LIN {X 0,Y 153.008,Z 595.327,A -85,B 0,C 180,E1 -24135.997,E2 -24135.997} C_VEL
LIN {X 0,Y 157.01,Z 598.55,A -85,B 0,C 180,E1 -24140.983,E2 -24140.983} C_VEL
LIN {X 0,Y 162.458,Z 600.625,A -85,B 0,C 180,E1 -24145.633,E2 -24145.633} C_VEL
LIN {X 0,Y 169.132,Z 601.557,A -85,B 0,C 180,E1 -24149.91,E2 -24149.91} C_VEL
LIN {X 0,Y 176.931,Z 601.358,A -85,B 0,C 180,E1 -24153.787,E2 -24153.787} C_VEL
LIN {X 0,Y 185.752,Z 600.036,A -85,B 0,C 180,E1 -24157.255,E2 -24157.255} C_VEL
LIN {X 0,Y 195.529,Z 597.531,A -85,B 0,C 180,E1 -24160.314,E2 -24160.314} C_VEL
LIN {X 0,Y 197.725,Z 596.972,A -85,B 0,C 180,E1 -24161.717,E2 -24161.717} C_VEL
LIN {X 0,Y 197.721,Z 597.127,A -85,B 0,C 180,E1 -24162.481,E2 -24162.481} C_VEL
LIN {X 0,Y 196.64,Z 597.978,A -85,B 0,C 180,E1 -24164.372,E2 -24164.372} C_VEL
LIN {X 0,Y 193.625,Z 599.675,A -85,B 0,C 180,E1 -24166.398,E2 -24166.398} C_VEL
LIN {X 0,Y 192.66,Z 600.123,A -85,B 0,C 180,E1 -24166.851,E2 -24166.851} C_VEL
LIN {X 0,Y 184.258,Z 603.417,A -85,B 0,C 180,E1 -24169.577,E2 -24169.577} C_VEL
LIN {X 0,Y 175.235,Z 606.225,A -85,B 0,C 180,E1 -24173.015,E2 -24173.015} C_VEL
LIN {X 0,Y 167.435,Z 608.021,A -85,B 0,C 180,E1 -24176.929,E2 -24176.929} C_VEL
LIN {X 0,Y 160.889,Z 608.807,A -85,B 0,C 180,E1 -24181.281,E2 -24181.281} C_VEL
LIN {X 0,Y 155.776,Z 608.587,A -85,B 0,C 180,E1 -24186.043,E2 -24186.043} C_VEL
LIN {X 0,Y 151.98,Z 607.326,A -85,B 0,C 180,E1 -24191.113,E2 -24191.113} C_VEL
LIN {X 0,Y 149.998,Z 605.016,A -85,B 0,C 180,E1 -24196.451,E2 -24196.451} C_VEL
LIN {X 0,Y 149.476,Z 601.54,A -85,B 0,C 180,E1 -24201.891,E2 -24201.891} C_VEL
LIN {X 0,Y 150.246,Z 596.672,A -85,B 0,C 180,E1 -24207.319,E2 -24207.319} C_VEL
LIN {X 0,Y 150.489,Z 593.443,A -85,B 0,C 180,E1 -24210,E2 -24210} C_VEL
LIN {X 0,Y 150.474,Z 587.289,A -85,B 0,C 180,E1 -24214.017,E2 -24214.017} C_VEL
LIN {X 0,Y 150.541,Z 579.575,A -85,B 0,C 180,E1 -24218.051,E2 -24218.051} C_VEL
LIN {X 0,Y 151.009,Z 570.809,A -85,B 0,C 180,E1 -24221.807,E2 -24221.807} C_VEL
LIN {X 0,Y 151.993,Z 560.329,A -85,B 0,C 180,E1 -24225.419,E2 -24225.419} C_VEL
LIN {X 0,Y 152.344,Z 554.548,A -85,B 0,C 180,E1 -24227.103,E2 -24227.103} C_VEL
LIN {X 0,Y 150.807,Z 542.716,A -85,B 0,C 180,E1 -24229.913,E2 -24229.913} C_VEL
LIN {X 0,Y 149.592,Z 528.841,A -85,B 0,C 180,E1 -24232.622,E2 -24232.622} C_VEL
LIN {X 0,Y 149.049,Z 513.657,A -85,B 0,C 180,E1 -24234.924,E2 -24234.924} C_VEL
LIN {X 0,Y 149.125,Z 509.454,A -85,B 0,C 180,E1 -24235.449,E2 -24235.449} C_VEL
LIN {X 0,Y 150.143,Z 505.621,A -85,B 0,C 180,E1 -24240.99,E2 -24240.99} C_VEL
LIN {X 0,Y 151.273,Z 502.439,A -85,B 0,C 180,E1 -24245.531,E2 -24245.531} C_VEL
LIN {X 0,Y 151.527,Z 500.732,A -85,B 0,C 180,E1 -24247.957,E2 -24247.957} C_VEL
LIN {X 0,Y 150.881,Z 497.692,A -85,B 0,C 180,E1 -24252.599,E2 -24252.599} C_VEL
LIN {X 0,Y 150.453,Z 497.743,A -85,B 0,C 180,E1 -24254.085,E2 -24254.085} C_VEL
LIN {X 0,Y 148.952,Z 497.931,A -85,B 0,C 180,E1 -24256.277,E2 -24256.277} C_VEL
LIN {X 0,Y 143.472,Z 498.608,A -85,B 0,C 180,E1 -24263.01,E2 -24263.01} C_VEL
LIN {X 0,Y 143.122,Z 498.65,A -85,B 0,C 180,E1 -24264.606,E2 -24264.606} C_VEL
LIN {X 0,Y 143.186,Z 498.648,A -85,B 0,C 180,E1 -24267.323,E2 -24267.323} C_VEL
LIN {X 0,Y 143.19,Z 498.642,A -85,B 0,C 180,E1 -24272.063,E2 -24272.063} C_VEL
LIN {X 0,Y 143.278,Z 498.634,A -85,B 0,C 180,E1 -24278.745,E2 -24278.745} C_VEL
LIN {X 0,Y 143.324,Z 498.632,A -85,B 0,C 180,E1 -24282.89,E2 -24282.89} C_VEL
LIN {X 0,Y 143.603,Z 498.591,A -85,B 0,C 180,E1 -24288.711,E2 -24288.711} C_VEL
LIN {X 0,Y 143.686,Z 498.585,A -85,B 0,C 180,E1 -24291.563,E2 -24291.563} C_VEL
LIN {X 0,Y 144.179,Z 498.523,A -85,B 0,C 180,E1 -24300,E2 -24300} C_VEL
LIN {X 0,Y 143.686,Z 498.584,A -85,B 0,C 180,E1 -24308.438,E2 -24308.438} C_VEL
LIN {X 0,Y 143.572,Z 498.6,A -85,B 0,C 180,E1 -24311.758,E2 -24311.758} C_VEL
LIN {X 0,Y 143.307,Z 498.631,A -85,B 0,C 180,E1 -24317.113,E2 -24317.113} C_VEL
LIN {X 0,Y 143.278,Z 498.636,A -85,B 0,C 180,E1 -24321.255,E2 -24321.255} C_VEL
LIN {X 0,Y 143.192,Z 498.648,A -85,B 0,C 180,E1 -24327.938,E2 -24327.938} C_VEL
LIN {X 0,Y 143.145,Z 498.647,A -85,B 0,C 180,E1 -24333.421,E2 -24333.421} C_VEL
LIN {X 0,Y 143.062,Z 498.663,A -85,B 0,C 180,E1 -24339.691,E2 -24339.691} C_VEL
LIN {X 0,Y 143.057,Z 498.661,A -85,B 0,C 180,E1 -24343.456,E2 -24343.456} C_VEL
LIN {X 0,Y 143.069,Z 498.662,A -85,B 0,C 180,E1 -24347.465,E2 -24347.465} C_VEL
LIN {X 0,Y 143.108,Z 498.654,A -85,B 0,C 180,E1 -24351.792,E2 -24351.792} C_VEL
LIN {X 0,Y 143.188,Z 498.646,A -85,B 0,C 180,E1 -24357.323,E2 -24357.323} C_VEL
LIN {X 0,Y 143.193,Z 498.647,A -85,B 0,C 180,E1 -24362.063,E2 -24362.063} C_VEL
LIN {X 0,Y 143.28,Z 498.633,A -85,B 0,C 180,E1 -24368.746,E2 -24368.746} C_VEL
LIN {X 0,Y 143.305,Z 498.633,A -85,B 0,C 180,E1 -24372.887,E2 -24372.887} C_VEL
LIN {X 0,Y 143.54,Z 498.603,A -85,B 0,C 180,E1 -24378.706,E2 -24378.706} C_VEL
LIN {X 0,Y 143.627,Z 498.594,A -85,B 0,C 180,E1 -24381.559,E2 -24381.559} C_VEL
LIN {X 0,Y 144.179,Z 498.527,A -85,B 0,C 180,E1 -24390,E2 -24390} C_VEL
LIN {X 0,Y 143.63,Z 498.594,A -85,B 0,C 180,E1 -24398.442,E2 -24398.442} C_VEL
LIN {X 0,Y 143.509,Z 498.606,A -85,B 0,C 180,E1 -24401.631,E2 -24401.631} C_VEL
LIN {X 0,Y 143.305,Z 498.633,A -85,B 0,C 180,E1 -24407.113,E2 -24407.113} C_VEL
LIN {X 0,Y 143.28,Z 498.633,A -85,B 0,C 180,E1 -24411.255,E2 -24411.255} C_VEL
LIN {X 0,Y 143.194,Z 498.647,A -85,B 0,C 180,E1 -24417.938,E2 -24417.938} C_VEL
LIN {X 0,Y 143.172,Z 498.649,A -85,B 0,C 180,E1 -24423.436,E2 -24423.436} C_VEL
LIN {X 0,Y 143.078,Z 498.657,A -85,B 0,C 180,E1 -24429.685,E2 -24429.685} C_VEL
LIN {X 0,Y 143.059,Z 498.665,A -85,B 0,C 180,E1 -24433.454,E2 -24433.454} C_VEL
LIN {X 0,Y 143.019,Z 498.665,A -85,B 0,C 180,E1 -24437.486,E2 -24437.486} C_VEL
LIN {X 0,Y 142.933,Z 498.682,A -85,B 0,C 180,E1 -24441.881,E2 -24441.881} C_VEL
LIN {X 0,Y 142.658,Z 498.708,A -85,B 0,C 180,E1 -24447.185,E2 -24447.185} C_VEL
LIN {X 0,Y 142.204,Z 498.771,A -85,B 0,C 180,E1 -24453.589,E2 -24453.589} C_VEL
LIN {X 0,Y 142.169,Z 498.848,A -85,B 0,C 180,E1 -24455.785,E2 -24455.785} C_VEL
LIN {X 0,Y 144.366,Z 512.297,A -85,B 0,C 180,E1 -24457.963,E2 -24457.963} C_VEL
LIN {X 0,Y 146.228,Z 522.624,A -85,B 0,C 180,E1 -24459.99,E2 -24459.99} C_VEL
LIN {X 0,Y 146.161,Z 525.789,A -85,B 0,C 180,E1 -24460.696,E2 -24460.696} C_VEL
LIN {X 0,Y 144.531,Z 538.8,A -85,B 0,C 180,E1 -24464.125,E2 -24464.125} C_VEL
LIN {X 0,Y 143.248,Z 550.554,A -85,B 0,C 180,E1 -24467.964,E2 -24467.964} C_VEL
LIN {X 0,Y 142.27,Z 561.149,A -85,B 0,C 180,E1 -24472.268,E2 -24472.268} C_VEL
LIN {X 0,Y 141.759,Z 570.856,A -85,B 0,C 180,E1 -24477.158,E2 -24477.158} C_VEL
LIN {X 0,Y 141.689,Z 577.811,A -85,B 0,C 180,E1 -24481.421,E2 -24481.421} C_VEL
LIN {X 0,Y 142.098,Z 583.58,A -85,B 0,C 180,E1 -24485.676,E2 -24485.676} C_VEL
LIN {X 0,Y 143.502,Z 590.092,A -85,B 0,C 180,E1 -24491.619,E2 -24491.619} C_VEL
LIN {X 0,Y 146.244,Z 594.625,A -85,B 0,C 180,E1 -24496.758,E2 -24496.758} C_VEL
LIN {X 0,Y 150.409,Z 598.253,A -85,B 0,C 180,E1 -24501.95,E2 -24501.95} C_VEL
LIN {X 0,Y 156.095,Z 600.718,A -85,B 0,C 180,E1 -24506.759,E2 -24506.759} C_VEL
LIN {X 0,Y 163.032,Z 602.071,A -85,B 0,C 180,E1 -24511.151,E2 -24511.151} C_VEL
LIN {X 0,Y 171.146,Z 602.303,A -85,B 0,C 180,E1 -24515.093,E2 -24515.093} C_VEL
LIN {X 0,Y 180.244,Z 601.445,A -85,B 0,C 180,E1 -24518.599,E2 -24518.599} C_VEL
LIN {X 0,Y 190.21,Z 599.482,A -85,B 0,C 180,E1 -24521.688,E2 -24521.688} C_VEL
LIN {X 0,Y 190.811,Z 599.467,A -85,B 0,C 180,E1 -24522.553,E2 -24522.553} C_VEL
LIN {X 0,Y 188.352,Z 600.781,A -85,B 0,C 180,E1 -24524.85,E2 -24524.85} C_VEL
LIN {X 0,Y 183.913,Z 602.443,A -85,B 0,C 180,E1 -24526.54,E2 -24526.54} C_VEL
LIN {X 0,Y 174.157,Z 605.288,A -85,B 0,C 180,E1 -24529.784,E2 -24529.784} C_VEL
LIN {X 0,Y 165.429,Z 607.134,A -85,B 0,C 180,E1 -24533.503,E2 -24533.503} C_VEL
LIN {X 0,Y 157.935,Z 608.004,A -85,B 0,C 180,E1 -24537.724,E2 -24537.724} C_VEL
LIN {X 0,Y 151.845,Z 607.905,A -85,B 0,C 180,E1 -24542.429,E2 -24542.429} C_VEL
LIN {X 0,Y 147.187,Z 606.83,A -85,B 0,C 180,E1 -24547.543,E2 -24547.543} C_VEL
LIN {X 0,Y 144.13,Z 604.743,A -85,B 0,C 180,E1 -24552.988,E2 -24552.988} C_VEL
LIN {X 0,Y 142.804,Z 601.556,A -85,B 0,C 180,E1 -24558.646,E2 -24558.646} C_VEL
LIN {X 0,Y 142.978,Z 597.154,A -85,B 0,C 180,E1 -24564.358,E2 -24564.358} C_VEL
LIN {X 0,Y 143.527,Z 594.379,A -85,B 0,C 180,E1 -24567.193,E2 -24567.193} C_VEL
LIN {X 0,Y 143.742,Z 590.953,A -85,B 0,C 180,E1 -24570,E2 -24570} C_VEL
LIN {X 0,Y 143.679,Z 585.695,A -85,B 0,C 180,E1 -24573.505,E2 -24573.505} C_VEL
LIN {X 0,Y 143.696,Z 579.205,A -85,B 0,C 180,E1 -24577.023,E2 -24577.023} C_VEL
LIN {X 0,Y 144.117,Z 569.784,A -85,B 0,C 180,E1 -24581.248,E2 -24581.248} C_VEL
LIN {X 0,Y 145.163,Z 558.179,A -85,B 0,C 180,E1 -24585.443,E2 -24585.443} C_VEL
LIN {X 0,Y 145.4,Z 554.724,A -85,B 0,C 180,E1 -24586.497,E2 -24586.497} C_VEL
LIN {X 0,Y 143.724,Z 542.198,A -85,B 0,C 180,E1 -24589.644,E2 -24589.644} C_VEL
LIN {X 0,Y 142.532,Z 529.062,A -85,B 0,C 180,E1 -24592.361,E2 -24592.361} C_VEL
LIN {X 0,Y 141.964,Z 514.809,A -85,B 0,C 180,E1 -24594.689,E2 -24594.689} C_VEL
LIN {X 0,Y 142.057,Z 508.996,A -85,B 0,C 180,E1 -24595.553,E2 -24595.553} C_VEL
LIN {X 0,Y 143.396,Z 504.379,A -85,B 0,C 180,E1 -24602.624,E2 -24602.624} C_VEL
LIN {X 0,Y 144.212,Z 502.265,A -85,B 0,C 180,E1 -24605.789,E2 -24605.789} C_VEL
LIN {X 0,Y 144.426,Z 501.307,A -85,B 0,C 180,E1 -24607.224,E2 -24607.224} C_VEL
LIN {X 0,Y 143.911,Z 498.562,A -85,B 0,C 180,E1 -24611.532,E2 -24611.532} C_VEL
LIN {X 0,Y 143.428,Z 498.618,A -85,B 0,C 180,E1 -24617.307,E2 -24617.307} C_VEL
LIN {X 0,Y 143.146,Z 498.649,A -85,B 0,C 180,E1 -24623.903,E2 -24623.903} C_VEL
LIN {X 0,Y 143.122,Z 498.65,A -85,B 0,C 180,E1 -24624.606,E2 -24624.606} C_VEL
LIN {X 0,Y 142.413,Z 498.746,A -85,B 0,C 180,E1 -24626.956,E2 -24626.956} C_VEL
LIN {X 0,Y 140.803,Z 498.943,A -85,B 0,C 180,E1 -24629.272,E2 -24629.272} C_VEL
LIN {X 0,Y 137.111,Z 499.403,A -85,B 0,C 180,E1 -24634.004,E2 -24634.004} C_VEL
LIN {X 0,Y 136.163,Z 499.525,A -85,B 0,C 180,E1 -24636.497,E2 -24636.497} C_VEL
LIN {X 0,Y 136.127,Z 499.523,A -85,B 0,C 180,E1 -24637.341,E2 -24637.341} C_VEL
LIN {X 0,Y 136.258,Z 499.508,A -85,B 0,C 180,E1 -24641.973,E2 -24641.973} C_VEL
LIN {X 0,Y 136.502,Z 499.477,A -85,B 0,C 180,E1 -24648.116,E2 -24648.116} C_VEL
LIN {X 0,Y 136.61,Z 499.467,A -85,B 0,C 180,E1 -24651.122,E2 -24651.122} C_VEL
LIN {X 0,Y 137.136,Z 499.4,A -85,B 0,C 180,E1 -24660.001,E2 -24660.001} C_VEL
LIN {X 0,Y 136.61,Z 499.467,A -85,B 0,C 180,E1 -24668.879,E2 -24668.879} C_VEL
LIN {X 0,Y 136.493,Z 499.483,A -85,B 0,C 180,E1 -24671.957,E2 -24671.957} C_VEL
LIN {X 0,Y 136.246,Z 499.512,A -85,B 0,C 180,E1 -24678.03,E2 -24678.03} C_VEL
LIN {X 0,Y 136.199,Z 499.518,A -85,B 0,C 180,E1 -24681.75,E2 -24681.75} C_VEL
LIN {X 0,Y 136.118,Z 499.53,A -85,B 0,C 180,E1 -24688.629,E2 -24688.629} C_VEL
LIN {X 0,Y 136.044,Z 499.536,A -85,B 0,C 180,E1 -24694.63,E2 -24694.63} C_VEL
LIN {X 0,Y 136.033,Z 499.538,A -85,B 0,C 180,E1 -24699.199,E2 -24699.199} C_VEL
LIN {X 0,Y 135.999,Z 499.541,A -85,B 0,C 180,E1 -24703.658,E2 -24703.658} C_VEL
LIN {X 0,Y 136.033,Z 499.54,A -85,B 0,C 180,E1 -24707.807,E2 -24707.807} C_VEL
LIN {X 0,Y 136.057,Z 499.532,A -85,B 0,C 180,E1 -24711.695,E2 -24711.695} C_VEL
LIN {X 0,Y 136.092,Z 499.533,A -85,B 0,C 180,E1 -24715.718,E2 -24715.718} C_VEL
LIN {X 0,Y 136.149,Z 499.526,A -85,B 0,C 180,E1 -24722.317,E2 -24722.317} C_VEL
LIN {X 0,Y 136.247,Z 499.509,A -85,B 0,C 180,E1 -24728.834,E2 -24728.834} C_VEL
LIN {X 0,Y 136.272,Z 499.507,A -85,B 0,C 180,E1 -24735.057,E2 -24735.057} C_VEL
LIN {X 0,Y 136.447,Z 499.484,A -85,B 0,C 180,E1 -24738.138,E2 -24738.138} C_VEL
LIN {X 0,Y 136.553,Z 499.475,A -85,B 0,C 180,E1 -24741.118,E2 -24741.118} C_VEL
LIN {X 0,Y 137.136,Z 499.404,A -85,B 0,C 180,E1 -24750,E2 -24750} C_VEL
LIN {X 0,Y 136.555,Z 499.474,A -85,B 0,C 180,E1 -24758.882,E2 -24758.882} C_VEL
LIN {X 0,Y 136.444,Z 499.484,A -85,B 0,C 180,E1 -24761.89,E2 -24761.89} C_VEL
LIN {X 0,Y 136.246,Z 499.514,A -85,B 0,C 180,E1 -24768.03,E2 -24768.03} C_VEL
LIN {X 0,Y 136.201,Z 499.513,A -85,B 0,C 180,E1 -24771.749,E2 -24771.749} C_VEL
LIN {X 0,Y 136.104,Z 499.528,A -85,B 0,C 180,E1 -24778.617,E2 -24778.617} C_VEL
LIN {X 0,Y 136.082,Z 499.533,A -85,B 0,C 180,E1 -24784.618,E2 -24784.618} C_VEL
LIN {X 0,Y 136.053,Z 499.532,A -85,B 0,C 180,E1 -24789.208,E2 -24789.208} C_VEL
LIN {X 0,Y 135.999,Z 499.545,A -85,B 0,C 180,E1 -24793.657,E2 -24793.657} C_VEL
LIN {X 0,Y 135.961,Z 499.543,A -85,B 0,C 180,E1 -24797.779,E2 -24797.779} C_VEL
LIN {X 0,Y 135.888,Z 499.558,A -85,B 0,C 180,E1 -24801.637,E2 -24801.637} C_VEL
LIN {X 0,Y 135.657,Z 499.581,A -85,B 0,C 180,E1 -24805.988,E2 -24805.988} C_VEL
LIN {X 0,Y 135.188,Z 499.647,A -85,B 0,C 180,E1 -24812.102,E2 -24812.102} C_VEL
LIN {X 0,Y 135.129,Z 499.65,A -85,B 0,C 180,E1 -24815.897,E2 -24815.897} C_VEL
LIN {X 0,Y 137.922,Z 516.294,A -85,B 0,C 180,E1 -24818.882,E2 -24818.882} C_VEL
LIN {X 0,Y 139.254,Z 523.712,A -85,B 0,C 180,E1 -24820.466,E2 -24820.466} C_VEL
LIN {X 0,Y 137.75,Z 536.019,A -85,B 0,C 180,E1 -24823.703,E2 -24823.703} C_VEL
LIN {X 0,Y 136.451,Z 547.152,A -85,B 0,C 180,E1 -24827.355,E2 -24827.355} C_VEL
LIN {X 0,Y 135.402,Z 558.315,A -85,B 0,C 180,E1 -24831.873,E2 -24831.873} C_VEL
LIN {X 0,Y 134.91,Z 567.261,A -85,B 0,C 180,E1 -24836.266,E2 -24836.266} C_VEL
LIN {X 0,Y 134.818,Z 573.635,A -85,B 0,C 180,E1 -24839.999,E2 -24839.999} C_VEL
LIN {X 0,Y 135.041,Z 580.054,A -85,B 0,C 180,E1 -24844.477,E2 -24844.477} C_VEL
LIN {X 0,Y 135.991,Z 586.675,A -85,B 0,C 180,E1 -24850.019,E2 -24850.019} C_VEL
LIN {X 0,Y 138.585,Z 592.587,A -85,B 0,C 180,E1 -24856.195,E2 -24856.195} C_VEL
LIN {X 0,Y 141.542,Z 595.948,A -85,B 0,C 180,E1 -24860.339,E2 -24860.339} C_VEL
LIN {X 0,Y 146.668,Z 599.355,A -85,B 0,C 180,E1 -24865.547,E2 -24865.547} C_VEL
LIN {X 0,Y 153.253,Z 601.654,A -85,B 0,C 180,E1 -24870.294,E2 -24870.294} C_VEL
LIN {X 0,Y 161.114,Z 602.867,A -85,B 0,C 180,E1 -24874.546,E2 -24874.546} C_VEL
LIN {X 0,Y 170.016,Z 602.999,A -85,B 0,C 180,E1 -24878.32,E2 -24878.32} C_VEL
LIN {X 0,Y 179.888,Z 602.056,A -85,B 0,C 180,E1 -24881.618,E2 -24881.618} C_VEL
LIN {X 0,Y 182.895,Z 601.722,A -85,B 0,C 180,E1 -24883.104,E2 -24883.104} C_VEL
LIN {X 0,Y 178.839,Z 603.077,A -85,B 0,C 180,E1 -24884.979,E2 -24884.979} C_VEL
LIN {X 0,Y 168.804,Z 605.434,A -85,B 0,C 180,E1 -24888.229,E2 -24888.229} C_VEL
LIN {X 0,Y 159.802,Z 606.846,A -85,B 0,C 180,E1 -24891.996,E2 -24891.996} C_VEL
LIN {X 0,Y 151.763,Z 607.311,A -85,B 0,C 180,E1 -24896.466,E2 -24896.466} C_VEL
LIN {X 0,Y 145.644,Z 606.854,A -85,B 0,C 180,E1 -24901.148,E2 -24901.148} C_VEL
LIN {X 0,Y 140.773,Z 605.448,A -85,B 0,C 180,E1 -24906.459,E2 -24906.459} C_VEL
LIN {X 0,Y 137.543,Z 603.026,A -85,B 0,C 180,E1 -24912.146,E2 -24912.146} C_VEL
LIN {X 0,Y 136.054,Z 598.966,A -85,B 0,C 180,E1 -24918.949,E2 -24918.949} C_VEL
LIN {X 0,Y 136.299,Z 594.862,A -85,B 0,C 180,E1 -24924.08,E2 -24924.08} C_VEL
LIN {X 0,Y 136.862,Z 591.94,A -85,B 0,C 180,E1 -24927.056,E2 -24927.056} C_VEL
LIN {X 0,Y 137.023,Z 588.289,A -85,B 0,C 180,E1 -24930,E2 -24930} C_VEL
LIN {X 0,Y 136.982,Z 582.68,A -85,B 0,C 180,E1 -24933.677,E2 -24933.677} C_VEL
LIN {X 0,Y 136.988,Z 574.415,A -85,B 0,C 180,E1 -24938.11,E2 -24938.11} C_VEL
LIN {X 0,Y 137.403,Z 565.912,A -85,B 0,C 180,E1 -24941.806,E2 -24941.806} C_VEL
LIN {X 0,Y 138.405,Z 554.702,A -85,B 0,C 180,E1 -24945.8,E2 -24945.8} C_VEL
LIN {X 0,Y 136.981,Z 543.992,A -85,B 0,C 180,E1 -24948.703,E2 -24948.703} C_VEL
LIN {X 0,Y 135.712,Z 531.069,A -85,B 0,C 180,E1 -24951.612,E2 -24951.612} C_VEL
LIN {X 0,Y 134.973,Z 518,A -85,B 0,C 180,E1 -24954.003,E2 -24954.003} C_VEL
LIN {X 0,Y 134.986,Z 508.64,A -85,B 0,C 180,E1 -24955.438,E2 -24955.438} C_VEL
LIN {X 0,Y 136.32,Z 504.122,A -85,B 0,C 180,E1 -24962.774,E2 -24962.774} C_VEL
LIN {X 0,Y 137.173,Z 502.018,A -85,B 0,C 180,E1 -24966.138,E2 -24966.138} C_VEL
LIN {X 0,Y 137.245,Z 500.905,A -85,B 0,C 180,E1 -24967.915,E2 -24967.915} C_VEL
LIN {X 0,Y 136.935,Z 499.431,A -85,B 0,C 180,E1 -24970.407,E2 -24970.407} C_VEL
LIN {X 0,Y 136.452,Z 499.488,A -85,B 0,C 180,E1 -24976.143,E2 -24976.143} C_VEL
LIN {X 0,Y 136.167,Z 499.518,A -85,B 0,C 180,E1 -24981.731,E2 -24981.731} C_VEL
LIN {X 0,Y 136.096,Z 499.531,A -85,B 0,C 180,E1 -24985.714,E2 -24985.714} C_VEL
LIN {X 0,Y 136.146,Z 499.52,A -85,B 0,C 180,E1 -24992.317,E2 -24992.317} C_VEL
LIN {X 0,Y 136.127,Z 499.523,A -85,B 0,C 180,E1 -24997.341,E2 -24997.341} C_VEL
LIN {X 0,Y 135.629,Z 499.591,A -85,B 0,C 180,E1 -24999.812,E2 -24999.812} C_VEL
LIN {X 0,Y 134.228,Z 499.773,A -85,B 0,C 180,E1 -25002.258,E2 -25002.258} C_VEL
LIN {X 0,Y 129.908,Z 500.307,A -85,B 0,C 180,E1 -25008.981,E2 -25008.981} C_VEL
LIN {X 0,Y 129.524,Z 500.346,A -85,B 0,C 180,E1 -25010.752,E2 -25010.752} C_VEL
LIN {X 0,Y 130.091,Z 500.277,A -85,B 0,C 180,E1 -25020.001,E2 -25020.001} C_VEL
LIN {X 0,Y 129.532,Z 500.348,A -85,B 0,C 180,E1 -25029.368,E2 -25029.368} C_VEL
LIN {X 0,Y 129.394,Z 500.366,A -85,B 0,C 180,E1 -25032.549,E2 -25032.549} C_VEL
LIN {X 0,Y 129.157,Z 500.396,A -85,B 0,C 180,E1 -25039.056,E2 -25039.056} C_VEL
LIN {X 0,Y 129.109,Z 500.399,A -85,B 0,C 180,E1 -25042.399,E2 -25042.399} C_VEL
LIN {X 0,Y 129.037,Z 500.411,A -85,B 0,C 180,E1 -25049.374,E2 -25049.374} C_VEL
LIN {X 0,Y 128.96,Z 500.419,A -85,B 0,C 180,E1 -25055.169,E2 -25055.169} C_VEL
LIN {X 0,Y 128.935,Z 500.418,A -85,B 0,C 180,E1 -25060.852,E2 -25060.852} C_VEL
LIN {X 0,Y 128.923,Z 500.425,A -85,B 0,C 180,E1 -25065.128,E2 -25065.128} C_VEL
LIN {X 0,Y 128.959,Z 500.416,A -85,B 0,C 180,E1 -25069.728,E2 -25069.728} C_VEL
LIN {X 0,Y 128.994,Z 500.416,A -85,B 0,C 180,E1 -25074.811,E2 -25074.811} C_VEL
LIN {X 0,Y 129.036,Z 500.408,A -85,B 0,C 180,E1 -25080.647,E2 -25080.647} C_VEL
LIN {X 0,Y 129.111,Z 500.396,A -85,B 0,C 180,E1 -25087.602,E2 -25087.602} C_VEL
LIN {X 0,Y 129.156,Z 500.395,A -85,B 0,C 180,E1 -25090.945,E2 -25090.945} C_VEL
LIN {X 0,Y 129.369,Z 500.364,A -85,B 0,C 180,E1 -25097.923,E2 -25097.923} C_VEL
LIN {X 0,Y 129.479,Z 500.356,A -85,B 0,C 180,E1 -25100.629,E2 -25100.629} C_VEL
LIN {X 0,Y 130.091,Z 500.281,A -85,B 0,C 180,E1 -25110,E2 -25110} C_VEL
LIN {X 0,Y 129.481,Z 500.356,A -85,B 0,C 180,E1 -25119.372,E2 -25119.372} C_VEL
LIN {X 0,Y 129.347,Z 500.366,A -85,B 0,C 180,E1 -25122.553,E2 -25122.553} C_VEL
LIN {X 0,Y 129.157,Z 500.395,A -85,B 0,C 180,E1 -25129.056,E2 -25129.056} C_VEL
LIN {X 0,Y 129.111,Z 500.396,A -85,B 0,C 180,E1 -25132.398,E2 -25132.398} C_VEL
LIN {X 0,Y 129.039,Z 500.408,A -85,B 0,C 180,E1 -25139.373,E2 -25139.373} C_VEL
LIN {X 0,Y 128.995,Z 500.416,A -85,B 0,C 180,E1 -25145.189,E2 -25145.189} C_VEL
LIN {X 0,Y 128.953,Z 500.417,A -85,B 0,C 180,E1 -25150.845,E2 -25150.845} C_VEL
LIN {X 0,Y 128.915,Z 500.426,A -85,B 0,C 180,E1 -25155.131,E2 -25155.131} C_VEL
LIN {X 0,Y 128.851,Z 500.43,A -85,B 0,C 180,E1 -25159.784,E2 -25159.784} C_VEL
LIN {X 0,Y 128.641,Z 500.459,A -85,B 0,C 180,E1 -25165.035,E2 -25165.035} C_VEL
LIN {X 0,Y 128.18,Z 500.518,A -85,B 0,C 180,E1 -25171.315,E2 -25171.315} C_VEL
LIN {X 0,Y 128.1,Z 500.545,A -85,B 0,C 180,E1 -25176.176,E2 -25176.176} C_VEL
LIN {X 0,Y 130.435,Z 514.22,A -85,B 0,C 180,E1 -25178.672,E2 -25178.672} C_VEL
LIN {X 0,Y 132.042,Z 522.98,A -85,B 0,C 180,E1 -25180.569,E2 -25180.569} C_VEL
LIN {X 0,Y 130.886,Z 534.1,A -85,B 0,C 180,E1 -25183.626,E2 -25183.626} C_VEL
LIN {X 0,Y 129.473,Z 546.18,A -85,B 0,C 180,E1 -25187.709,E2 -25187.709} C_VEL
LIN {X 0,Y 128.466,Z 557.428,A -85,B 0,C 180,E1 -25192.418,E2 -25192.418} C_VEL
LIN {X 0,Y 128.043,Z 566.099,A -85,B 0,C 180,E1 -25196.853,E2 -25196.853} C_VEL
LIN {X 0,Y 127.958,Z 572.573,A -85,B 0,C 180,E1 -25200.786,E2 -25200.786} C_VEL
LIN {X 0,Y 128.341,Z 580.211,A -85,B 0,C 180,E1 -25206.287,E2 -25206.287} C_VEL
LIN {X 0,Y 129.764,Z 587.161,A -85,B 0,C 180,E1 -25212.511,E2 -25212.511} C_VEL
LIN {X 0,Y 132.846,Z 592.772,A -85,B 0,C 180,E1 -25218.507,E2 -25218.507} C_VEL
LIN {X 0,Y 137.388,Z 597.118,A -85,B 0,C 180,E1 -25224.156,E2 -25224.156} C_VEL
LIN {X 0,Y 143.57,Z 600.352,A -85,B 0,C 180,E1 -25229.309,E2 -25229.309} C_VEL
LIN {X 0,Y 151.093,Z 602.529,A -85,B 0,C 180,E1 -25233.929,E2 -25233.929} C_VEL
LIN {X 0,Y 159.801,Z 603.643,A -85,B 0,C 180,E1 -25238.004,E2 -25238.004} C_VEL
LIN {X 0,Y 169.49,Z 603.71,A -85,B 0,C 180,E1 -25241.563,E2 -25241.563} C_VEL
LIN {X 0,Y 173.82,Z 603.52,A -85,B 0,C 180,E1 -25243.298,E2 -25243.298} C_VEL
LIN {X 0,Y 163.577,Z 605.412,A -85,B 0,C 180,E1 -25246.572,E2 -25246.572} C_VEL
LIN {X 0,Y 154.285,Z 606.384,A -85,B 0,C 180,E1 -25250.377,E2 -25250.377} C_VEL
LIN {X 0,Y 145.75,Z 606.434,A -85,B 0,C 180,E1 -25255.058,E2 -25255.058} C_VEL
LIN {X 0,Y 139.555,Z 605.644,A -85,B 0,C 180,E1 -25259.761,E2 -25259.761} C_VEL
LIN {X 0,Y 134.444,Z 603.904,A -85,B 0,C 180,E1 -25265.279,E2 -25265.279} C_VEL
LIN {X 0,Y 131.029,Z 601.2,A -85,B 0,C 180,E1 -25271.226,E2 -25271.226} C_VEL
LIN {X 0,Y 129.473,Z 597.264,A -85,B 0,C 180,E1 -25277.705,E2 -25277.705} C_VEL
LIN {X 0,Y 129.699,Z 592.413,A -85,B 0,C 180,E1 -25283.778,E2 -25283.778} C_VEL
LIN {X 0,Y 130.238,Z 589.325,A -85,B 0,C 180,E1 -25286.906,E2 -25286.906} C_VEL
LIN {X 0,Y 130.367,Z 585.481,A -85,B 0,C 180,E1 -25290,E2 -25290} C_VEL
LIN {X 0,Y 130.252,Z 579.485,A -85,B 0,C 180,E1 -25293.867,E2 -25293.867} C_VEL
LIN {X 0,Y 130.299,Z 570.655,A -85,B 0,C 180,E1 -25298.53,E2 -25298.53} C_VEL
LIN {X 0,Y 130.905,Z 559.932,A -85,B 0,C 180,E1 -25303.114,E2 -25303.114} C_VEL
LIN {X 0,Y 131.416,Z 553.21,A -85,B 0,C 180,E1 -25305.509,E2 -25305.509} C_VEL
LIN {X 0,Y 129.566,Z 540.521,A -85,B 0,C 180,E1 -25308.993,E2 -25308.993} C_VEL
LIN {X 0,Y 128.327,Z 527.464,A -85,B 0,C 180,E1 -25311.962,E2 -25311.962} C_VEL
LIN {X 0,Y 127.801,Z 513.007,A -85,B 0,C 180,E1 -25314.574,E2 -25314.574} C_VEL
LIN {X 0,Y 127.917,Z 508.243,A -85,B 0,C 180,E1 -25315.31,E2 -25315.31} C_VEL
LIN {X 0,Y 129.23,Z 503.862,A -85,B 0,C 180,E1 -25322.945,E2 -25322.945} C_VEL
LIN {X 0,Y 130.093,Z 501.79,A -85,B 0,C 180,E1 -25326.459,E2 -25326.459} C_VEL
LIN {X 0,Y 129.978,Z 500.297,A -85,B 0,C 180,E1 -25329.194,E2 -25329.194} C_VEL
LIN {X 0,Y 129.486,Z 500.354,A -85,B 0,C 180,E1 -25335.123,E2 -25335.123} C_VEL
LIN {X 0,Y 129.164,Z 500.394,A -85,B 0,C 180,E1 -25339.619,E2 -25339.619} C_VEL
LIN {X 0,Y 129.037,Z 500.409,A -85,B 0,C 180,E1 -25344.783,E2 -25344.783} C_VEL
LIN {X 0,Y 129.033,Z 500.406,A -85,B 0,C 180,E1 -25350.647,E2 -25350.647} C_VEL
LIN {X 0,Y 129.109,Z 500.401,A -85,B 0,C 180,E1 -25357.602,E2 -25357.602} C_VEL
LIN {X 0,Y 129.164,Z 500.39,A -85,B 0,C 180,E1 -25360.946,E2 -25360.946} C_VEL
LIN {X 0,Y 129.419,Z 500.36,A -85,B 0,C 180,E1 -25367.815,E2 -25367.815} C_VEL
LIN {X 0,Y 129.524,Z 500.346,A -85,B 0,C 180,E1 -25370.752,E2 -25370.752} C_VEL
LIN {X 0,Y 128.778,Z 500.445,A -85,B 0,C 180,E1 -25373.359,E2 -25373.359} C_VEL
LIN {X 0,Y 127.232,Z 500.634,A -85,B 0,C 180,E1 -25375.937,E2 -25375.937} C_VEL
LIN {X 0,Y 122.848,Z 501.182,A -85,B 0,C 180,E1 -25383.05,E2 -25383.05} C_VEL
LIN {X 0,Y 122.484,Z 501.217,A -85,B 0,C 180,E1 -25384.927,E2 -25384.927} C_VEL
LIN {X 0,Y 122.458,Z 501.23,A -85,B 0,C 180,E1 -25389.915,E2 -25389.915} C_VEL
LIN {X 0,Y 122.264,Z 501.252,A -85,B 0,C 180,E1 -25393.294,E2 -25393.294} C_VEL
LIN {X 0,Y 122.048,Z 501.283,A -85,B 0,C 180,E1 -25400.213,E2 -25400.213} C_VEL
LIN {X 0,Y 121.985,Z 501.284,A -85,B 0,C 180,E1 -25403.785,E2 -25403.785} C_VEL
LIN {X 0,Y 121.94,Z 501.295,A -85,B 0,C 180,E1 -25410.172,E2 -25410.172} C_VEL
LIN {X 0,Y 121.885,Z 501.302,A -85,B 0,C 180,E1 -25416.172,E2 -25416.172} C_VEL
LIN {X 0,Y 121.873,Z 501.297,A -85,B 0,C 180,E1 -25421.439,E2 -25421.439} C_VEL
LIN {X 0,Y 121.886,Z 501.299,A -85,B 0,C 180,E1 -25428.556,E2 -25428.556} C_VEL
LIN {X 0,Y 121.947,Z 501.294,A -85,B 0,C 180,E1 -25434.809,E2 -25434.809} C_VEL
LIN {X 0,Y 121.944,Z 501.288,A -85,B 0,C 180,E1 -25439.827,E2 -25439.827} C_VEL
LIN {X 0,Y 121.986,Z 501.286,A -85,B 0,C 180,E1 -25446.216,E2 -25446.216} C_VEL
LIN {X 0,Y 122.048,Z 501.278,A -85,B 0,C 180,E1 -25449.788,E2 -25449.788} C_VEL
LIN {X 0,Y 122.242,Z 501.25,A -85,B 0,C 180,E1 -25456.705,E2 -25456.705} C_VEL
LIN {X 0,Y 122.408,Z 501.237,A -85,B 0,C 180,E1 -25460.082,E2 -25460.082} C_VEL
LIN {X 0,Y 122.598,Z 501.209,A -85,B 0,C 180,E1 -25466.714,E2 -25466.714} C_VEL
LIN {X 0,Y 123.044,Z 501.159,A -85,B 0,C 180,E1 -25470,E2 -25470} C_VEL
LIN {X 0,Y 122.429,Z 501.233,A -85,B 0,C 180,E1 -25476.593,E2 -25476.593} C_VEL
LIN {X 0,Y 122.321,Z 501.241,A -85,B 0,C 180,E1 -25482.377,E2 -25482.377} C_VEL
LIN {X 0,Y 122.112,Z 501.273,A -85,B 0,C 180,E1 -25486.725,E2 -25486.725} C_VEL
LIN {X 0,Y 122.027,Z 501.279,A -85,B 0,C 180,E1 -25492.851,E2 -25492.851} C_VEL
LIN {X 0,Y 121.953,Z 501.294,A -85,B 0,C 180,E1 -25497.454,E2 -25497.454} C_VEL
LIN {X 0,Y 121.914,Z 501.291,A -85,B 0,C 180,E1 -25501.254,E2 -25501.254} C_VEL
LIN {X 0,Y 121.915,Z 501.298,A -85,B 0,C 180,E1 -25506.189,E2 -25506.189} C_VEL
LIN {X 0,Y 121.886,Z 501.299,A -85,B 0,C 180,E1 -25511.444,E2 -25511.444} C_VEL
LIN {X 0,Y 121.806,Z 501.309,A -85,B 0,C 180,E1 -25516.18,E2 -25516.18} C_VEL
LIN {X 0,Y 121.752,Z 501.317,A -85,B 0,C 180,E1 -25520.582,E2 -25520.582} C_VEL
LIN {X 0,Y 121.617,Z 501.334,A -85,B 0,C 180,E1 -25524.697,E2 -25524.697} C_VEL
LIN {X 0,Y 121.172,Z 501.391,A -85,B 0,C 180,E1 -25530.46,E2 -25530.46} C_VEL
LIN {X 0,Y 121.093,Z 501.398,A -85,B 0,C 180,E1 -25536.521,E2 -25536.521} C_VEL
LIN {X 0,Y 123.514,Z 515.3,A -85,B 0,C 180,E1 -25539.228,E2 -25539.228} C_VEL
LIN {X 0,Y 124.995,Z 523.585,A -85,B 0,C 180,E1 -25541.137,E2 -25541.137} C_VEL
LIN {X 0,Y 123.515,Z 535.74,A -85,B 0,C 180,E1 -25544.743,E2 -25544.743} C_VEL
LIN {X 0,Y 122.4,Z 546.454,A -85,B 0,C 180,E1 -25548.615,E2 -25548.615} C_VEL
LIN {X 0,Y 121.526,Z 557.029,A -85,B 0,C 180,E1 -25553.358,E2 -25553.358} C_VEL
LIN {X 0,Y 121.185,Z 566.212,A -85,B 0,C 180,E1 -25558.338,E2 -25558.338} C_VEL
LIN {X 0,Y 121.206,Z 573.847,A -85,B 0,C 180,E1 -25563.324,E2 -25563.324} C_VEL
LIN {X 0,Y 121.857,Z 580.191,A -85,B 0,C 180,E1 -25568.29,E2 -25568.29} C_VEL
LIN {X 0,Y 123.891,Z 587.701,A -85,B 0,C 180,E1 -25575.34,E2 -25575.34} C_VEL
LIN {X 0,Y 128.478,Z 594.055,A -85,B 0,C 180,E1 -25582.514,E2 -25582.514} C_VEL
LIN {X 0,Y 134.066,Z 598.204,A -85,B 0,C 180,E1 -25588.151,E2 -25588.151} C_VEL
LIN {X 0,Y 141.19,Z 601.312,A -85,B 0,C 180,E1 -25593.198,E2 -25593.198} C_VEL
LIN {X 0,Y 149.649,Z 603.381,A -85,B 0,C 180,E1 -25597.627,E2 -25597.627} C_VEL
LIN {X 0,Y 161.275,Z 604.523,A -85,B 0,C 180,E1 -25602.198,E2 -25602.198} C_VEL
LIN {X 0,Y 163.716,Z 604.585,A -85,B 0,C 180,E1 -25603.132,E2 -25603.132} C_VEL
LIN {X 0,Y 153.565,Z 605.571,A -85,B 0,C 180,E1 -25606.647,E2 -25606.647} C_VEL
LIN {X 0,Y 144.589,Z 605.692,A -85,B 0,C 180,E1 -25610.81,E2 -25610.81} C_VEL
LIN {X 0,Y 136.865,Z 604.967,A -85,B 0,C 180,E1 -25615.608,E2 -25615.608} C_VEL
LIN {X 0,Y 130.675,Z 603.353,A -85,B 0,C 180,E1 -25621.05,E2 -25621.05} C_VEL
LIN {X 0,Y 126.133,Z 600.791,A -85,B 0,C 180,E1 -25627.043,E2 -25627.043} C_VEL
LIN {X 0,Y 123.541,Z 597.288,A -85,B 0,C 180,E1 -25633.474,E2 -25633.474} C_VEL
LIN {X 0,Y 122.842,Z 592.657,A -85,B 0,C 180,E1 -25640.117,E2 -25640.117} C_VEL
LIN {X 0,Y 123.394,Z 588.231,A -85,B 0,C 180,E1 -25645.099,E2 -25645.099} C_VEL
LIN {X 0,Y 123.768,Z 584.586,A -85,B 0,C 180,E1 -25648.373,E2 -25648.373} C_VEL
LIN {X 0,Y 123.641,Z 578.812,A -85,B 0,C 180,E1 -25652.443,E2 -25652.443} C_VEL
LIN {X 0,Y 123.531,Z 570.069,A -85,B 0,C 180,E1 -25657.354,E2 -25657.354} C_VEL
LIN {X 0,Y 123.886,Z 561.188,A -85,B 0,C 180,E1 -25661.452,E2 -25661.452} C_VEL
LIN {X 0,Y 124.498,Z 552.405,A -85,B 0,C 180,E1 -25664.844,E2 -25664.844} C_VEL
LIN {X 0,Y 122.617,Z 540.212,A -85,B 0,C 180,E1 -25668.375,E2 -25668.375} C_VEL
LIN {X 0,Y 121.314,Z 527.267,A -85,B 0,C 180,E1 -25671.51,E2 -25671.51} C_VEL
LIN {X 0,Y 120.76,Z 513.041,A -85,B 0,C 180,E1 -25674.269,E2 -25674.269} C_VEL
LIN {X 0,Y 120.849,Z 507.844,A -85,B 0,C 180,E1 -25675.167,E2 -25675.167} C_VEL
LIN {X 0,Y 122.157,Z 503.548,A -85,B 0,C 180,E1 -25683.131,E2 -25683.131} C_VEL
LIN {X 0,Y 122.986,Z 501.167,A -85,B 0,C 180,E1 -25687.497,E2 -25687.497} C_VEL
LIN {X 0,Y 122.655,Z 501.208,A -85,B 0,C 180,E1 -25691.851,E2 -25691.851} C_VEL
LIN {X 0,Y 122.143,Z 501.271,A -85,B 0,C 180,E1 -25698.418,E2 -25698.418} C_VEL
LIN {X 0,Y 121.988,Z 501.287,A -85,B 0,C 180,E1 -25704.822,E2 -25704.822} C_VEL
LIN {X 0,Y 121.942,Z 501.292,A -85,B 0,C 180,E1 -25709.826,E2 -25709.826} C_VEL
LIN {X 0,Y 121.984,Z 501.29,A -85,B 0,C 180,E1 -25716.216,E2 -25716.216} C_VEL
LIN {X 0,Y 122.052,Z 501.275,A -85,B 0,C 180,E1 -25719.789,E2 -25719.789} C_VEL
LIN {X 0,Y 122.266,Z 501.253,A -85,B 0,C 180,E1 -25726.708,E2 -25726.708} C_VEL
LIN {X 0,Y 122.427,Z 501.226,A -85,B 0,C 180,E1 -25730.694,E2 -25730.694} C_VEL
LIN {X 0,Y 123.045,Z 501.155,A -85,B 0,C 180,E1 -25740.001,E2 -25740.001} C_VEL
LIN {X 0,Y 122.484,Z 501.217,A -85,B 0,C 180,E1 -25744.927,E2 -25744.927} C_VEL
LIN {X 0,Y 121.69,Z 501.322,A -85,B 0,C 180,E1 -25747.668,E2 -25747.668} C_VEL
LIN {X 0,Y 119.998,Z 501.538,A -85,B 0,C 180,E1 -25750.369,E2 -25750.369} C_VEL
LIN {X 0,Y 115.26,Z 502.125,A -85,B 0,C 180,E1 -25757.873,E2 -25757.873} C_VEL
LIN {X 0,Y 114.936,Z 502.158,A -85,B 0,C 180,E1 -25759.872,E2 -25759.872} C_VEL
LIN {X 0,Y 114.875,Z 502.171,A -85,B 0,C 180,E1 -25765.358,E2 -25765.358} C_VEL
LIN {X 0,Y 114.862,Z 502.173,A -85,B 0,C 180,E1 -25771.063,E2 -25771.063} C_VEL
LIN {X 0,Y 114.781,Z 502.187,A -85,B 0,C 180,E1 -25777.757,E2 -25777.757} C_VEL
LIN {X 0,Y 114.788,Z 502.181,A -85,B 0,C 180,E1 -25782.718,E2 -25782.718} C_VEL
LIN {X 0,Y 114.804,Z 502.184,A -85,B 0,C 180,E1 -25787.671,E2 -25787.671} C_VEL
LIN {X 0,Y 114.814,Z 502.182,A -85,B 0,C 180,E1 -25792.728,E2 -25792.728} C_VEL
LIN {X 0,Y 114.871,Z 502.168,A -85,B 0,C 180,E1 -25798.932,E2 -25798.932} C_VEL
LIN {X 0,Y 114.949,Z 502.162,A -85,B 0,C 180,E1 -25806.508,E2 -25806.508} C_VEL
LIN {X 0,Y 115.014,Z 502.159,A -85,B 0,C 180,E1 -25812.21,E2 -25812.21} C_VEL
LIN {X 0,Y 115.254,Z 502.121,A -85,B 0,C 180,E1 -25817.334,E2 -25817.334} C_VEL
LIN {X 0,Y 115.366,Z 502.113,A -85,B 0,C 180,E1 -25823.002,E2 -25823.002} C_VEL
LIN {X 0,Y 115.996,Z 502.037,A -85,B 0,C 180,E1 -25830,E2 -25830} C_VEL
LIN {X 0,Y 115.369,Z 502.112,A -85,B 0,C 180,E1 -25836.998,E2 -25836.998} C_VEL
LIN {X 0,Y 115.255,Z 502.121,A -85,B 0,C 180,E1 -25842.667,E2 -25842.667} C_VEL
LIN {X 0,Y 115.015,Z 502.159,A -85,B 0,C 180,E1 -25847.79,E2 -25847.79} C_VEL
LIN {X 0,Y 114.95,Z 502.161,A -85,B 0,C 180,E1 -25853.493,E2 -25853.493} C_VEL
LIN {X 0,Y 114.872,Z 502.168,A -85,B 0,C 180,E1 -25861.068,E2 -25861.068} C_VEL
LIN {X 0,Y 114.805,Z 502.18,A -85,B 0,C 180,E1 -25867.747,E2 -25867.747} C_VEL
LIN {X 0,Y 114.794,Z 502.185,A -85,B 0,C 180,E1 -25872.719,E2 -25872.719} C_VEL
LIN {X 0,Y 114.737,Z 502.186,A -85,B 0,C 180,E1 -25877.639,E2 -25877.639} C_VEL
LIN {X 0,Y 114.59,Z 502.211,A -85,B 0,C 180,E1 -25882.875,E2 -25882.875} C_VEL
LIN {X 0,Y 114.164,Z 502.262,A -85,B 0,C 180,E1 -25889.526,E2 -25889.526} C_VEL
LIN {X 0,Y 114.086,Z 502.272,A -85,B 0,C 180,E1 -25896.868,E2 -25896.868} C_VEL
LIN {X 0,Y 116.951,Z 518.088,A -85,B 0,C 180,E1 -25900.243,E2 -25900.243} C_VEL
LIN {X 0,Y 117.794,Z 522.367,A -85,B 0,C 180,E1 -25901.295,E2 -25901.295} C_VEL
LIN {X 0,Y 116.952,Z 531.63,A -85,B 0,C 180,E1 -25904.05,E2 -25904.05} C_VEL
LIN {X 0,Y 115.586,Z 544.22,A -85,B 0,C 180,E1 -25908.712,E2 -25908.712} C_VEL
LIN {X 0,Y 114.692,Z 555.413,A -85,B 0,C 180,E1 -25913.843,E2 -25913.843} C_VEL
LIN {X 0,Y 114.384,Z 564.886,A -85,B 0,C 180,E1 -25919.119,E2 -25919.119} C_VEL
LIN {X 0,Y 114.518,Z 572.599,A -85,B 0,C 180,E1 -25924.399,E2 -25924.399} C_VEL
LIN {X 0,Y 115.439,Z 580.142,A -85,B 0,C 180,E1 -25930.523,E2 -25930.523} C_VEL
LIN {X 0,Y 117.812,Z 587.083,A -85,B 0,C 180,E1 -25937.353,E2 -25937.353} C_VEL
LIN {X 0,Y 122.05,Z 592.807,A -85,B 0,C 180,E1 -25943.77,E2 -25943.77} C_VEL
LIN {X 0,Y 127.9,Z 597.368,A -85,B 0,C 180,E1 -25949.639,E2 -25949.639} C_VEL
LIN {X 0,Y 135.325,Z 600.85,A -85,B 0,C 180,E1 -25954.839,E2 -25954.839} C_VEL
LIN {X 0,Y 144.09,Z 603.341,A -85,B 0,C 180,E1 -25959.351,E2 -25959.351} C_VEL
LIN {X 0,Y 152.233,Z 604.662,A -85,B 0,C 180,E1 -25962.615,E2 -25962.615} C_VEL
LIN {X 0,Y 152,Z 604.854,A -85,B 0,C 180,E1 -25963.502,E2 -25963.502} C_VEL
LIN {X 0,Y 143.71,Z 604.895,A -85,B 0,C 180,E1 -25966.791,E2 -25966.791} C_VEL
LIN {X 0,Y 135.004,Z 604.215,A -85,B 0,C 180,E1 -25971.34,E2 -25971.34} C_VEL
LIN {X 0,Y 127.717,Z 602.709,A -85,B 0,C 180,E1 -25976.613,E2 -25976.613} C_VEL
LIN {X 0,Y 122.098,Z 600.297,A -85,B 0,C 180,E1 -25982.581,E2 -25982.581} C_VEL
LIN {X 0,Y 118.249,Z 596.942,A -85,B 0,C 180,E1 -25989.108,E2 -25989.108} C_VEL
LIN {X 0,Y 116.489,Z 592.623,A -85,B 0,C 180,E1 -25996.035,E2 -25996.035} C_VEL
LIN {X 0,Y 116.667,Z 587.052,A -85,B 0,C 180,E1 -26003.08,E2 -26003.08} C_VEL
LIN {X 0,Y 117.196,Z 582.572,A -85,B 0,C 180,E1 -26007.422,E2 -26007.422} C_VEL
LIN {X 0,Y 117.091,Z 577.917,A -85,B 0,C 180,E1 -26010.859,E2 -26010.859} C_VEL
LIN {X 0,Y 116.824,Z 569.342,A -85,B 0,C 180,E1 -26016.043,E2 -26016.043} C_VEL
LIN {X 0,Y 117.035,Z 560.621,A -85,B 0,C 180,E1 -26020.378,E2 -26020.378} C_VEL
LIN {X 0,Y 117.632,Z 552.28,A -85,B 0,C 180,E1 -26023.826,E2 -26023.826} C_VEL
LIN {X 0,Y 115.814,Z 540.827,A -85,B 0,C 180,E1 -26027.387,E2 -26027.387} C_VEL
LIN {X 0,Y 114.336,Z 527.174,A -85,B 0,C 180,E1 -26030.933,E2 -26030.933} C_VEL
LIN {X 0,Y 113.703,Z 511.877,A -85,B 0,C 180,E1 -26034.085,E2 -26034.085} C_VEL
LIN {X 0,Y 113.785,Z 507.405,A -85,B 0,C 180,E1 -26034.95,E2 -26034.95} C_VEL
LIN {X 0,Y 115.081,Z 503.219,A -85,B 0,C 180,E1 -26043.341,E2 -26043.341} C_VEL
LIN {X 0,Y 115.623,Z 502.083,A -85,B 0,C 180,E1 -26045.806,E2 -26045.806} C_VEL
LIN {X 0,Y 115.944,Z 502.044,A -85,B 0,C 180,E1 -26048.001,E2 -26048.001} C_VEL
LIN {X 0,Y 115.477,Z 502.098,A -85,B 0,C 180,E1 -26053.087,E2 -26053.087} C_VEL
LIN {X 0,Y 115.124,Z 502.144,A -85,B 0,C 180,E1 -26057.816,E2 -26057.816} C_VEL
LIN {X 0,Y 114.959,Z 502.158,A -85,B 0,C 180,E1 -26062.632,E2 -26062.632} C_VEL
LIN {X 0,Y 114.87,Z 502.174,A -85,B 0,C 180,E1 -26068.931,E2 -26068.931} C_VEL
LIN {X 0,Y 114.947,Z 502.167,A -85,B 0,C 180,E1 -26076.508,E2 -26076.508} C_VEL
LIN {X 0,Y 115.021,Z 502.154,A -85,B 0,C 180,E1 -26082.212,E2 -26082.212} C_VEL
LIN {X 0,Y 115.287,Z 502.12,A -85,B 0,C 180,E1 -26087.258,E2 -26087.258} C_VEL
LIN {X 0,Y 115.394,Z 502.104,A -85,B 0,C 180,E1 -26089.473,E2 -26089.473} C_VEL
LIN {X 0,Y 115.538,Z 502.088,A -85,B 0,C 180,E1 -26096.513,E2 -26096.513} C_VEL
LIN {X 0,Y 115.997,Z 502.033,A -85,B 0,C 180,E1 -26100.001,E2 -26100.001} C_VEL
LIN {X 0,Y 115.392,Z 502.104,A -85,B 0,C 180,E1 -26107.104,E2 -26107.104} C_VEL
LIN {X 0,Y 115.287,Z 502.122,A -85,B 0,C 180,E1 -26112.743,E2 -26112.743} C_VEL
LIN {X 0,Y 114.936,Z 502.158,A -85,B 0,C 180,E1 -26119.872,E2 -26119.872} C_VEL
LIN {X 0,Y 114.231,Z 502.254,A -85,B 0,C 180,E1 -26122.792,E2 -26122.792} C_VEL
LIN {X 0,Y 112.582,Z 502.462,A -85,B 0,C 180,E1 -26125.673,E2 -26125.673} C_VEL
LIN {X 0,Y 107.957,Z 503.03,A -85,B 0,C 180,E1 -26133.704,E2 -26133.704} C_VEL
LIN {X 0,Y 107.711,Z 503.066,A -85,B 0,C 180,E1 -26135.842,E2 -26135.842} C_VEL
LIN {X 0,Y 107.682,Z 503.065,A -85,B 0,C 180,E1 -26140.744,E2 -26140.744} C_VEL
LIN {X 0,Y 107.683,Z 503.072,A -85,B 0,C 180,E1 -26145.884,E2 -26145.884} C_VEL
LIN {X 0,Y 107.709,Z 503.062,A -85,B 0,C 180,E1 -26151.538,E2 -26151.538} C_VEL
LIN {X 0,Y 107.809,Z 503.048,A -85,B 0,C 180,E1 -26158.567,E2 -26158.567} C_VEL
LIN {X 0,Y 107.913,Z 503.037,A -85,B 0,C 180,E1 -26166.999,E2 -26166.999} C_VEL
LIN {X 0,Y 108.033,Z 503.024,A -85,B 0,C 180,E1 -26174.917,E2 -26174.917} C_VEL
LIN {X 0,Y 108.256,Z 502.998,A -85,B 0,C 180,E1 -26178.77,E2 -26178.77} C_VEL
LIN {X 0,Y 108.446,Z 502.97,A -85,B 0,C 180,E1 -26186.285,E2 -26186.285} C_VEL
LIN {X 0,Y 108.945,Z 502.915,A -85,B 0,C 180,E1 -26190,E2 -26190} C_VEL
LIN {X 0,Y 108.308,Z 502.992,A -85,B 0,C 180,E1 -26197.457,E2 -26197.457} C_VEL
LIN {X 0,Y 108.176,Z 503.002,A -85,B 0,C 180,E1 -26202.956,E2 -26202.956} C_VEL
LIN {X 0,Y 107.907,Z 503.042,A -85,B 0,C 180,E1 -26209.006,E2 -26209.006} C_VEL
LIN {X 0,Y 107.861,Z 503.047,A -85,B 0,C 180,E1 -26214.185,E2 -26214.185} C_VEL
LIN {X 0,Y 107.797,Z 503.052,A -85,B 0,C 180,E1 -26222.052,E2 -26222.052} C_VEL
LIN {X 0,Y 107.709,Z 503.062,A -85,B 0,C 180,E1 -26228.463,E2 -26228.463} C_VEL
LIN {X 0,Y 107.643,Z 503.074,A -85,B 0,C 180,E1 -26235.906,E2 -26235.906} C_VEL
LIN {X 0,Y 107.545,Z 503.088,A -85,B 0,C 180,E1 -26241.647,E2 -26241.647} C_VEL
LIN {X 0,Y 107.154,Z 503.133,A -85,B 0,C 180,E1 -26248.351,E2 -26248.351} C_VEL
LIN {X 0,Y 107.133,Z 503.138,A -85,B 0,C 180,E1 -26257.452,E2 -26257.452} C_VEL
LIN {X 0,Y 109.956,Z 518.381,A -85,B 0,C 180,E1 -26260.878,E2 -26260.878} C_VEL
LIN {X 0,Y 110.797,Z 522.98,A -85,B 0,C 180,E1 -26262.079,E2 -26262.079} C_VEL
LIN {X 0,Y 109.575,Z 533.784,A -85,B 0,C 180,E1 -26265.653,E2 -26265.653} C_VEL
LIN {X 0,Y 108.411,Z 546.074,A -85,B 0,C 180,E1 -26270.672,E2 -26270.672} C_VEL
LIN {X 0,Y 107.842,Z 555.409,A -85,B 0,C 180,E1 -26275.327,E2 -26275.327} C_VEL
LIN {X 0,Y 107.724,Z 564.717,A -85,B 0,C 180,E1 -26280.934,E2 -26280.934} C_VEL
LIN {X 0,Y 108.139,Z 573.628,A -85,B 0,C 180,E1 -26287.468,E2 -26287.468} C_VEL
LIN {X 0,Y 109.798,Z 581.747,A -85,B 0,C 180,E1 -26294.834,E2 -26294.834} C_VEL
LIN {X 0,Y 113.298,Z 588.477,A -85,B 0,C 180,E1 -26301.85,E2 -26301.85} C_VEL
LIN {X 0,Y 118.524,Z 593.975,A -85,B 0,C 180,E1 -26308.318,E2 -26308.318} C_VEL
LIN {X 0,Y 125.555,Z 598.37,A -85,B 0,C 180,E1 -26314.038,E2 -26314.038} C_VEL
LIN {X 0,Y 133.97,Z 601.76,A -85,B 0,C 180,E1 -26319.014,E2 -26319.014} C_VEL
LIN {X 0,Y 141.998,Z 603.85,A -85,B 0,C 180,E1 -26322.589,E2 -26322.589} C_VEL
LIN {X 0,Y 140.795,Z 603.99,A -85,B 0,C 180,E1 -26323.91,E2 -26323.91} C_VEL
LIN {X 0,Y 129.657,Z 602.819,A -85,B 0,C 180,E1 -26329.424,E2 -26329.424} C_VEL
LIN {X 0,Y 122.048,Z 600.926,A -85,B 0,C 180,E1 -26334.841,E2 -26334.841} C_VEL
LIN {X 0,Y 116.123,Z 598.213,A -85,B 0,C 180,E1 -26341.041,E2 -26341.041} C_VEL
LIN {X 0,Y 111.353,Z 593.546,A -85,B 0,C 180,E1 -26349.688,E2 -26349.688} C_VEL
LIN {X 0,Y 109.947,Z 588.662,A -85,B 0,C 180,E1 -26357.072,E2 -26357.072} C_VEL
LIN {X 0,Y 110.532,Z 582.356,A -85,B 0,C 180,E1 -26364.527,E2 -26364.527} C_VEL
LIN {X 0,Y 110.718,Z 578.238,A -85,B 0,C 180,E1 -26368.181,E2 -26368.181} C_VEL
LIN {X 0,Y 110.343,Z 571.551,A -85,B 0,C 180,E1 -26372.738,E2 -26372.738} C_VEL
LIN {X 0,Y 110.253,Z 561.623,A -85,B 0,C 180,E1 -26378.246,E2 -26378.246} C_VEL
LIN {X 0,Y 110.786,Z 551.62,A -85,B 0,C 180,E1 -26382.828,E2 -26382.828} C_VEL
LIN {X 0,Y 108.869,Z 539.955,A -85,B 0,C 180,E1 -26386.675,E2 -26386.675} C_VEL
LIN {X 0,Y 107.339,Z 526.648,A -85,B 0,C 180,E1 -26390.355,E2 -26390.355} C_VEL
LIN {X 0,Y 106.679,Z 512.356,A -85,B 0,C 180,E1 -26393.54,E2 -26393.54} C_VEL
LIN {X 0,Y 106.728,Z 507.031,A -85,B 0,C 180,E1 -26394.562,E2 -26394.562} C_VEL
LIN {X 0,Y 107.993,Z 503.028,A -85,B 0,C 180,E1 -26403.607,E2 -26403.607} C_VEL
LIN {X 0,Y 108.515,Z 502.968,A -85,B 0,C 180,E1 -26405.653,E2 -26405.653} C_VEL
LIN {X 0,Y 108.751,Z 502.941,A -85,B 0,C 180,E1 -26409.15,E2 -26409.15} C_VEL
LIN {X 0,Y 108.198,Z 503.006,A -85,B 0,C 180,E1 -26415.602,E2 -26415.602} C_VEL
LIN {X 0,Y 107.891,Z 503.04,A -85,B 0,C 180,E1 -26421.414,E2 -26421.414} C_VEL
LIN {X 0,Y 107.813,Z 503.054,A -85,B 0,C 180,E1 -26428.568,E2 -26428.568} C_VEL
LIN {X 0,Y 107.912,Z 503.042,A -85,B 0,C 180,E1 -26436.999,E2 -26436.999} C_VEL
LIN {X 0,Y 108.041,Z 503.027,A -85,B 0,C 180,E1 -26444.919,E2 -26444.919} C_VEL
LIN {X 0,Y 108.307,Z 502.986,A -85,B 0,C 180,E1 -26448.775,E2 -26448.775} C_VEL
LIN {X 0,Y 108.464,Z 502.97,A -85,B 0,C 180,E1 -26456.285,E2 -26456.285} C_VEL
LIN {X 0,Y 108.948,Z 502.911,A -85,B 0,C 180,E1 -26460.001,E2 -26460.001} C_VEL
LIN {X 0,Y 108.341,Z 502.984,A -85,B 0,C 180,E1 -26467.455,E2 -26467.455} C_VEL
LIN {X 0,Y 108.204,Z 503.004,A -85,B 0,C 180,E1 -26473.026,E2 -26473.026} C_VEL
LIN {X 0,Y 107.866,Z 503.042,A -85,B 0,C 180,E1 -26479.8,E2 -26479.8} C_VEL
LIN {X 0,Y 107.86,Z 503.042,A -85,B 0,C 180,E1 -26484.187,E2 -26484.187} C_VEL
LIN {X 0,Y 107.785,Z 503.052,A -85,B 0,C 180,E1 -26492.043,E2 -26492.043} C_VEL
LIN {X 0,Y 107.711,Z 503.066,A -85,B 0,C 180,E1 -26495.842,E2 -26495.842} C_VEL
LIN {X 0,Y 107.463,Z 503.11,A -85,B 0,C 180,E1 -26497.926,E2 -26497.926} C_VEL
LIN {X 0,Y 106.689,Z 503.214,A -85,B 0,C 180,E1 -26499.989,E2 -26499.989} C_VEL
LIN {X 0,Y 104.281,Z 503.51,A -85,B 0,C 180,E1 -26504.101,E2 -26504.101} C_VEL
LIN {X 0,Y 100.912,Z 503.907,A -85,B 0,C 180,E1 -26510.657,E2 -26510.657} C_VEL
LIN {X 0,Y 100.569,Z 503.942,A -85,B 0,C 180,E1 -26512.956,E2 -26512.956} C_VEL
LIN {X 0,Y 100.702,Z 503.939,A -85,B 0,C 180,E1 -26516.877,E2 -26516.877} C_VEL
LIN {X 0,Y 100.788,Z 503.929,A -85,B 0,C 180,E1 -26525.268,E2 -26525.268} C_VEL
LIN {X 0,Y 100.818,Z 503.922,A -85,B 0,C 180,E1 -26529.602,E2 -26529.602} C_VEL
LIN {X 0,Y 101.104,Z 503.883,A -85,B 0,C 180,E1 -26536.703,E2 -26536.703} C_VEL
LIN {X 0,Y 101.244,Z 503.874,A -85,B 0,C 180,E1 -26542.02,E2 -26542.02} C_VEL
LIN {X 0,Y 101.868,Z 503.797,A -85,B 0,C 180,E1 -26550,E2 -26550} C_VEL
LIN {X 0,Y 101.246,Z 503.873,A -85,B 0,C 180,E1 -26557.981,E2 -26557.981} C_VEL
LIN {X 0,Y 101.105,Z 503.882,A -85,B 0,C 180,E1 -26563.298,E2 -26563.298} C_VEL
LIN {X 0,Y 100.819,Z 503.922,A -85,B 0,C 180,E1 -26570.399,E2 -26570.399} C_VEL
LIN {X 0,Y 100.777,Z 503.93,A -85,B 0,C 180,E1 -26574.959,E2 -26574.959} C_VEL
LIN {X 0,Y 100.703,Z 503.938,A -85,B 0,C 180,E1 -26583.124,E2 -26583.124} C_VEL
LIN {X 0,Y 100.656,Z 503.939,A -85,B 0,C 180,E1 -26589.82,E2 -26589.82} C_VEL
LIN {X 0,Y 100.595,Z 503.953,A -85,B 0,C 180,E1 -26595.681,E2 -26595.681} C_VEL
LIN {X 0,Y 100.493,Z 503.965,A -85,B 0,C 180,E1 -26600.992,E2 -26600.992} C_VEL
LIN {X 0,Y 100.124,Z 504.005,A -85,B 0,C 180,E1 -26607.387,E2 -26607.387} C_VEL
LIN {X 0,Y 100.195,Z 504.004,A -85,B 0,C 180,E1 -26618.131,E2 -26618.131} C_VEL
LIN {X 0,Y 102.987,Z 518.599,A -85,B 0,C 180,E1 -26621.626,E2 -26621.626} C_VEL
LIN {X 0,Y 103.705,Z 521.835,A -85,B 0,C 180,E1 -26622.504,E2 -26622.504} C_VEL
LIN {X 0,Y 102.984,Z 529.835,A -85,B 0,C 180,E1 -26625.171,E2 -26625.171} C_VEL
LIN {X 0,Y 101.844,Z 541.803,A -85,B 0,C 180,E1 -26630.065,E2 -26630.065} C_VEL
LIN {X 0,Y 101.119,Z 553.465,A -85,B 0,C 180,E1 -26636.014,E2 -26636.014} C_VEL
LIN {X 0,Y 101.075,Z 563.065,A -85,B 0,C 180,E1 -26641.992,E2 -26641.992} C_VEL
LIN {X 0,Y 101.699,Z 572.087,A -85,B 0,C 180,E1 -26648.944,E2 -26648.944} C_VEL
LIN {X 0,Y 103.279,Z 579.56,A -85,B 0,C 180,E1 -26655.794,E2 -26655.794} C_VEL
LIN {X 0,Y 106.967,Z 586.633,A -85,B 0,C 180,E1 -26663.216,E2 -26663.216} C_VEL
LIN {X 0,Y 112.473,Z 592.494,A -85,B 0,C 180,E1 -26669.992,E2 -26669.992} C_VEL
LIN {X 0,Y 119.801,Z 597.311,A -85,B 0,C 180,E1 -26675.919,E2 -26675.919} C_VEL
LIN {X 0,Y 130.885,Z 601.846,A -85,B 0,C 180,E1 -26682.082,E2 -26682.082} C_VEL
LIN {X 0,Y 132.005,Z 602.192,A -85,B 0,C 180,E1 -26682.588,E2 -26682.588} C_VEL
LIN {X 0,Y 130.975,Z 602.254,A -85,B 0,C 180,E1 -26683.976,E2 -26683.976} C_VEL
LIN {X 0,Y 120.306,Z 600.183,A -85,B 0,C 180,E1 -26690.014,E2 -26690.014} C_VEL
LIN {X 0,Y 113.192,Z 597.57,A -85,B 0,C 180,E1 -26696.026,E2 -26696.026} C_VEL
LIN {X 0,Y 107.805,Z 594.085,A -85,B 0,C 180,E1 -26702.848,E2 -26702.848} C_VEL
LIN {X 0,Y 104.616,Z 589.728,A -85,B 0,C 180,E1 -26710.372,E2 -26710.372} C_VEL
LIN {X 0,Y 103.727,Z 582.668,A -85,B 0,C 180,E1 -26720.247,E2 -26720.247} C_VEL
LIN {X 0,Y 104.302,Z 578.107,A -85,B 0,C 180,E1 -26725.168,E2 -26725.168} C_VEL
LIN {X 0,Y 104.242,Z 574.645,A -85,B 0,C 180,E1 -26728.068,E2 -26728.068} C_VEL
LIN {X 0,Y 103.713,Z 567.557,A -85,B 0,C 180,E1 -26732.913,E2 -26732.913} C_VEL
LIN {X 0,Y 103.622,Z 558.89,A -85,B 0,C 180,E1 -26737.796,E2 -26737.796} C_VEL
LIN {X 0,Y 103.993,Z 550.731,A -85,B 0,C 180,E1 -26741.697,E2 -26741.697} C_VEL
LIN {X 0,Y 102.11,Z 539.852,A -85,B 0,C 180,E1 -26745.511,E2 -26745.511} C_VEL
LIN {X 0,Y 100.461,Z 526.711,A -85,B 0,C 180,E1 -26749.408,E2 -26749.408} C_VEL
LIN {X 0,Y 99.715,Z 512.872,A -85,B 0,C 180,E1 -26752.748,E2 -26752.748} C_VEL
LIN {X 0,Y 99.71,Z 506.647,A -85,B 0,C 180,E1 -26754.046,E2 -26754.046} C_VEL
LIN {X 0,Y 100.204,Z 503.997,A -85,B 0,C 180,E1 -26760.391,E2 -26760.391} C_VEL
LIN {X 0,Y 100.966,Z 503.903,A -85,B 0,C 180,E1 -26763.838,E2 -26763.838} C_VEL
LIN {X 0,Y 101.621,Z 503.829,A -85,B 0,C 180,E1 -26768.493,E2 -26768.493} C_VEL
LIN {X 0,Y 101.25,Z 503.868,A -85,B 0,C 180,E1 -26773.957,E2 -26773.957} C_VEL
LIN {X 0,Y 100.847,Z 503.918,A -85,B 0,C 180,E1 -26781.156,E2 -26781.156} C_VEL
LIN {X 0,Y 100.719,Z 503.94,A -85,B 0,C 180,E1 -26786.86,E2 -26786.86} C_VEL
LIN {X 0,Y 100.786,Z 503.931,A -85,B 0,C 180,E1 -26795.268,E2 -26795.268} C_VEL
LIN {X 0,Y 100.82,Z 503.919,A -85,B 0,C 180,E1 -26799.602,E2 -26799.602} C_VEL
LIN {X 0,Y 101.2,Z 503.873,A -85,B 0,C 180,E1 -26807.976,E2 -26807.976} C_VEL
LIN {X 0,Y 101.28,Z 503.868,A -85,B 0,C 180,E1 -26812.023,E2 -26812.023} C_VEL
LIN {X 0,Y 101.872,Z 503.792,A -85,B 0,C 180,E1 -26820.001,E2 -26820.001} C_VEL
LIN {X 0,Y 101.28,Z 503.864,A -85,B 0,C 180,E1 -26827.978,E2 -26827.978} C_VEL
LIN {X 0,Y 101.13,Z 503.885,A -85,B 0,C 180,E1 -26833.364,E2 -26833.364} C_VEL
LIN {X 0,Y 100.818,Z 503.927,A -85,B 0,C 180,E1 -26840.399,E2 -26840.399} C_VEL
LIN {X 0,Y 100.775,Z 503.925,A -85,B 0,C 180,E1 -26844.959,E2 -26844.959} C_VEL
LIN {X 0,Y 100.692,Z 503.934,A -85,B 0,C 180,E1 -26853.117,E2 -26853.117} C_VEL
LIN {X 0,Y 100.641,Z 503.945,A -85,B 0,C 180,E1 -26859.812,E2 -26859.812} C_VEL
LIN {X 0,Y 100.653,Z 503.947,A -85,B 0,C 180,E1 -26865.714,E2 -26865.714} C_VEL
LIN {X 0,Y 100.646,Z 503.941,A -85,B 0,C 180,E1 -26871.064,E2 -26871.064} C_VEL
LIN {X 0,Y 100.569,Z 503.942,A -85,B 0,C 180,E1 -26872.956,E2 -26872.956} C_VEL
LIN {X 0,Y 99.866,Z 504.044,A -85,B 0,C 180,E1 -26876.301,E2 -26876.301} C_VEL
LIN {X 0,Y 98.277,Z 504.243,A -85,B 0,C 180,E1 -26879.615,E2 -26879.615} C_VEL
LIN {X 0,Y 93.906,Z 504.781,A -85,B 0,C 180,E1 -26888.902,E2 -26888.902} C_VEL
LIN {X 0,Y 93.709,Z 504.803,A -85,B 0,C 180,E1 -26891.37,E2 -26891.37} C_VEL
LIN {X 0,Y 94.068,Z 504.759,A -85,B 0,C 180,E1 -26897.048,E2 -26897.048} C_VEL
LIN {X 0,Y 94.177,Z 504.754,A -85,B 0,C 180,E1 -26901.417,E2 -26901.417} C_VEL
LIN {X 0,Y 94.794,Z 504.678,A -85,B 0,C 180,E1 -26910,E2 -26910} C_VEL
LIN {X 0,Y 94.179,Z 504.754,A -85,B 0,C 180,E1 -26918.584,E2 -26918.584} C_VEL
LIN {X 0,Y 94.025,Z 504.764,A -85,B 0,C 180,E1 -26923.659,E2 -26923.659} C_VEL
LIN {X 0,Y 93.695,Z 504.806,A -85,B 0,C 180,E1 -26932.028,E2 -26932.028} C_VEL
LIN {X 0,Y 93.626,Z 504.822,A -85,B 0,C 180,E1 -26936.769,E2 -26936.769} C_VEL
LIN {X 0,Y 93.601,Z 504.826,A -85,B 0,C 180,E1 -26944.315,E2 -26944.315} C_VEL
LIN {X 0,Y 93.531,Z 504.834,A -85,B 0,C 180,E1 -26952.554,E2 -26952.554} C_VEL
LIN {X 0,Y 93.419,Z 504.84,A -85,B 0,C 180,E1 -26958.792,E2 -26958.792} C_VEL
LIN {X 0,Y 93.132,Z 504.877,A -85,B 0,C 180,E1 -26966.109,E2 -26966.109} C_VEL
LIN {X 0,Y 93.311,Z 504.863,A -85,B 0,C 180,E1 -26978.968,E2 -26978.968} C_VEL
LIN {X 0,Y 96.231,Z 519.637,A -85,B 0,C 180,E1 -26982.749,E2 -26982.749} C_VEL
LIN {X 0,Y 96.719,Z 522.6,A -85,B 0,C 180,E1 -26983.645,E2 -26983.645} C_VEL
LIN {X 0,Y 95.504,Z 534.639,A -85,B 0,C 180,E1 -26988.324,E2 -26988.324} C_VEL
LIN {X 0,Y 94.695,Z 545.652,A -85,B 0,C 180,E1 -26993.607,E2 -26993.607} C_VEL
LIN {X 0,Y 94.396,Z 554.916,A -85,B 0,C 180,E1 -26998.933,E2 -26998.933} C_VEL
LIN {X 0,Y 94.58,Z 562.639,A -85,B 0,C 180,E1 -27004.261,E2 -27004.261} C_VEL
LIN {X 0,Y 95.539,Z 571.666,A -85,B 0,C 180,E1 -27011.67,E2 -27011.67} C_VEL
LIN {X 0,Y 97.608,Z 579.037,A -85,B 0,C 180,E1 -27018.905,E2 -27018.905} C_VEL
LIN {X 0,Y 102.041,Z 586.235,A -85,B 0,C 180,E1 -27026.592,E2 -27026.592} C_VEL
LIN {X 0,Y 110.185,Z 593.538,A -85,B 0,C 180,E1 -27035.033,E2 -27035.033} C_VEL
LIN {X 0,Y 118.604,Z 598.187,A -85,B 0,C 180,E1 -27040.678,E2 -27040.678} C_VEL
LIN {X 0,Y 123.053,Z 600.122,A -85,B 0,C 180,E1 -27043.264,E2 -27043.264} C_VEL
LIN {X 0,Y 111.205,Z 596.833,A -85,B 0,C 180,E1 -27050.802,E2 -27050.802} C_VEL
LIN {X 0,Y 104.607,Z 593.505,A -85,B 0,C 180,E1 -27057.487,E2 -27057.487} C_VEL
LIN {X 0,Y 99.966,Z 589.282,A -85,B 0,C 180,E1 -27065.05,E2 -27065.05} C_VEL
LIN {X 0,Y 97.691,Z 584.109,A -85,B 0,C 180,E1 -27073.275,E2 -27073.275} C_VEL
LIN {X 0,Y 97.716,Z 577.628,A -85,B 0,C 180,E1 -27081.729,E2 -27081.729} C_VEL
LIN {X 0,Y 98.026,Z 574.658,A -85,B 0,C 180,E1 -27084.858,E2 -27084.858} C_VEL
LIN {X 0,Y 97.662,Z 569.417,A -85,B 0,C 180,E1 -27088.969,E2 -27088.969} C_VEL
LIN {X 0,Y 97.165,Z 561.473,A -85,B 0,C 180,E1 -27094.147,E2 -27094.147} C_VEL
LIN {X 0,Y 97.196,Z 550.886,A -85,B 0,C 180,E1 -27099.888,E2 -27099.888} C_VEL
LIN {X 0,Y 97.169,Z 548.57,A -85,B 0,C 180,E1 -27100.944,E2 -27100.944} C_VEL
LIN {X 0,Y 94.68,Z 535.231,A -85,B 0,C 180,E1 -27105.708,E2 -27105.708} C_VEL
LIN {X 0,Y 93.166,Z 521.336,A -85,B 0,C 180,E1 -27109.843,E2 -27109.843} C_VEL
LIN {X 0,Y 92.667,Z 508.476,A -85,B 0,C 180,E1 -27112.946,E2 -27112.946} C_VEL
LIN {X 0,Y 92.712,Z 506.232,A -85,B 0,C 180,E1 -27113.433,E2 -27113.433} C_VEL
LIN {X 0,Y 92.688,Z 504.937,A -85,B 0,C 180,E1 -27117.061,E2 -27117.061} C_VEL
LIN {X 0,Y 93.98,Z 504.775,A -85,B 0,C 180,E1 -27124.655,E2 -27124.655} C_VEL
LIN {X 0,Y 94.215,Z 504.748,A -85,B 0,C 180,E1 -27126.638,E2 -27126.638} C_VEL
LIN {X 0,Y 94.313,Z 504.736,A -85,B 0,C 180,E1 -27132.118,E2 -27132.118} C_VEL
LIN {X 0,Y 93.881,Z 504.791,A -85,B 0,C 180,E1 -27138.469,E2 -27138.469} C_VEL
LIN {X 0,Y 93.649,Z 504.818,A -85,B 0,C 180,E1 -27145.639,E2 -27145.639} C_VEL
LIN {X 0,Y 93.669,Z 504.815,A -85,B 0,C 180,E1 -27154.205,E2 -27154.205} C_VEL
LIN {X 0,Y 93.695,Z 504.812,A -85,B 0,C 180,E1 -27157.974,E2 -27157.974} C_VEL
LIN {X 0,Y 94.098,Z 504.76,A -85,B 0,C 180,E1 -27167.053,E2 -27167.053} C_VEL
LIN {X 0,Y 94.212,Z 504.748,A -85,B 0,C 180,E1 -27171.42,E2 -27171.42} C_VEL
LIN {X 0,Y 94.799,Z 504.673,A -85,B 0,C 180,E1 -27180.001,E2 -27180.001} C_VEL
LIN {X 0,Y 94.212,Z 504.746,A -85,B 0,C 180,E1 -27188.581,E2 -27188.581} C_VEL
LIN {X 0,Y 94.048,Z 504.766,A -85,B 0,C 180,E1 -27193.722,E2 -27193.722} C_VEL
LIN {X 0,Y 93.694,Z 504.811,A -85,B 0,C 180,E1 -27202.028,E2 -27202.028} C_VEL
LIN {X 0,Y 93.623,Z 504.821,A -85,B 0,C 180,E1 -27206.771,E2 -27206.771} C_VEL
LIN {X 0,Y 93.588,Z 504.821,A -85,B 0,C 180,E1 -27214.306,E2 -27214.306} C_VEL
LIN {X 0,Y 93.535,Z 504.827,A -85,B 0,C 180,E1 -27222.552,E2 -27222.552} C_VEL
LIN {X 0,Y 93.546,Z 504.828,A -85,B 0,C 180,E1 -27228.704,E2 -27228.704} C_VEL
LIN {X 0,Y 93.6,Z 504.826,A -85,B 0,C 180,E1 -27235.686,E2 -27235.686} C_VEL
LIN {X 0,Y 93.671,Z 504.817,A -85,B 0,C 180,E1 -27244.205,E2 -27244.205} C_VEL
LIN {X 0,Y 93.709,Z 504.803,A -85,B 0,C 180,E1 -27251.37,E2 -27251.37} C_VEL
LIN {X 0,Y 93.332,Z 504.867,A -85,B 0,C 180,E1 -27254.979,E2 -27254.979} C_VEL
LIN {X 0,Y 92.148,Z 505.025,A -85,B 0,C 180,E1 -27258.576,E2 -27258.576} C_VEL
LIN {X 0,Y 88.963,Z 505.418,A -85,B 0,C 180,E1 -27265.974,E2 -27265.974} C_VEL
LIN {X 0,Y 87.536,Z 505.573,A -85,B 0,C 180,E1 -27271.181,E2 -27271.181} C_VEL
LIN {X 0,Y 87.088,Z 505.637,A -85,B 0,C 180,E1 -27279.289,E2 -27279.289} C_VEL
LIN {X 0,Y 86.933,Z 505.648,A -85,B 0,C 180,E1 -27284.037,E2 -27284.037} C_VEL
LIN {X 0,Y 86.648,Z 505.691,A -85,B 0,C 180,E1 -27288.932,E2 -27288.932} C_VEL
LIN {X 0,Y 86.588,Z 505.699,A -85,B 0,C 180,E1 -27296.767,E2 -27296.767} C_VEL
LIN {X 0,Y 86.519,Z 505.708,A -85,B 0,C 180,E1 -27305.677,E2 -27305.677} C_VEL
LIN {X 0,Y 86.446,Z 505.716,A -85,B 0,C 180,E1 -27312.97,E2 -27312.97} C_VEL
LIN {X 0,Y 86.337,Z 505.723,A -85,B 0,C 180,E1 -27319.365,E2 -27319.365} C_VEL
LIN {X 0,Y 86.099,Z 505.756,A -85,B 0,C 180,E1 -27325.152,E2 -27325.152} C_VEL
LIN {X 0,Y 85.828,Z 505.787,A -85,B 0,C 180,E1 -27335.83,E2 -27335.83} C_VEL
LIN {X 0,Y 86.525,Z 505.887,A -85,B 0,C 180,E1 -27340.114,E2 -27340.114} C_VEL
LIN {X 0,Y 89.478,Z 520.22,A -85,B 0,C 180,E1 -27344.043,E2 -27344.043} C_VEL
LIN {X 0,Y 89.775,Z 522.165,A -85,B 0,C 180,E1 -27344.679,E2 -27344.679} C_VEL
LIN {X 0,Y 88.539,Z 535.485,A -85,B 0,C 180,E1 -27350.288,E2 -27350.288} C_VEL
LIN {X 0,Y 87.98,Z 545.282,A -85,B 0,C 180,E1 -27355.417,E2 -27355.417} C_VEL
LIN {X 0,Y 87.9,Z 554.374,A -85,B 0,C 180,E1 -27361.145,E2 -27361.145} C_VEL
LIN {X 0,Y 88.25,Z 562.088,A -85,B 0,C 180,E1 -27366.86,E2 -27366.86} C_VEL
LIN {X 0,Y 89.379,Z 569.862,A -85,B 0,C 180,E1 -27373.644,E2 -27373.644} C_VEL
LIN {X 0,Y 92.305,Z 578.505,A -85,B 0,C 180,E1 -27382.376,E2 -27382.376} C_VEL
LIN {X 0,Y 97.525,Z 585.7,A -85,B 0,C 180,E1 -27390.294,E2 -27390.294} C_VEL
LIN {X 0,Y 104.623,Z 591.76,A -85,B 0,C 180,E1 -27397.197,E2 -27397.197} C_VEL
LIN {X 0,Y 113.423,Z 596.849,A -85,B 0,C 180,E1 -27402.968,E2 -27402.968} C_VEL
LIN {X 0,Y 110.264,Z 595.951,A -85,B 0,C 180,E1 -27405.483,E2 -27405.483} C_VEL
LIN {X 0,Y 102.391,Z 592.789,A -85,B 0,C 180,E1 -27411.847,E2 -27411.847} C_VEL
LIN {X 0,Y 95.131,Z 587.559,A -85,B 0,C 180,E1 -27421.301,E2 -27421.301} C_VEL
LIN {X 0,Y 91.649,Z 580.892,A -85,B 0,C 180,E1 -27432.137,E2 -27432.137} C_VEL
LIN {X 0,Y 91.611,Z 574.075,A -85,B 0,C 180,E1 -27441.174,E2 -27441.174} C_VEL
LIN {X 0,Y 91.838,Z 571.266,A -85,B 0,C 180,E1 -27444.174,E2 -27444.174} C_VEL
LIN {X 0,Y 91.167,Z 565.252,A -85,B 0,C 180,E1 -27448.894,E2 -27448.894} C_VEL
LIN {X 0,Y 90.636,Z 556.663,A -85,B 0,C 180,E1 -27454.447,E2 -27454.447} C_VEL
LIN {X 0,Y 90.654,Z 548.563,A -85,B 0,C 180,E1 -27458.919,E2 -27458.919} C_VEL
LIN {X 0,Y 88.817,Z 539.456,A -85,B 0,C 180,E1 -27462.568,E2 -27462.568} C_VEL
LIN {X 0,Y 86.838,Z 526.428,A -85,B 0,C 180,E1 -27467.043,E2 -27467.043} C_VEL
LIN {X 0,Y 85.816,Z 512.568,A -85,B 0,C 180,E1 -27470.995,E2 -27470.995} C_VEL
LIN {X 0,Y 85.72,Z 505.809,A -85,B 0,C 180,E1 -27472.76,E2 -27472.76} C_VEL
LIN {X 0,Y 87.112,Z 505.632,A -85,B 0,C 180,E1 -27486.218,E2 -27486.218} C_VEL
LIN {X 0,Y 87.188,Z 505.626,A -85,B 0,C 180,E1 -27490.154,E2 -27490.154} C_VEL
LIN {X 0,Y 86.904,Z 505.659,A -85,B 0,C 180,E1 -27496.705,E2 -27496.705} C_VEL
LIN {X 0,Y 86.612,Z 505.695,A -85,B 0,C 180,E1 -27505.389,E2 -27505.389} C_VEL
LIN {X 0,Y 86.585,Z 505.695,A -85,B 0,C 180,E1 -27513.233,E2 -27513.233} C_VEL
LIN {X 0,Y 86.649,Z 505.684,A -85,B 0,C 180,E1 -27521.069,E2 -27521.069} C_VEL
LIN {X 0,Y 86.969,Z 505.651,A -85,B 0,C 180,E1 -27525.971,E2 -27525.971} C_VEL
LIN {X 0,Y 87.119,Z 505.628,A -85,B 0,C 180,E1 -27530.716,E2 -27530.716} C_VEL
LIN {X 0,Y 87.726,Z 505.554,A -85,B 0,C 180,E1 -27540.001,E2 -27540.001} C_VEL
LIN {X 0,Y 87.119,Z 505.632,A -85,B 0,C 180,E1 -27549.286,E2 -27549.286} C_VEL
LIN {X 0,Y 86.951,Z 505.647,A -85,B 0,C 180,E1 -27554.088,E2 -27554.088} C_VEL
LIN {X 0,Y 86.664,Z 505.69,A -85,B 0,C 180,E1 -27558.929,E2 -27558.929} C_VEL
LIN {X 0,Y 86.585,Z 505.698,A -85,B 0,C 180,E1 -27566.766,E2 -27566.766} C_VEL
LIN {X 0,Y 86.507,Z 505.707,A -85,B 0,C 180,E1 -27575.667,E2 -27575.667} C_VEL
LIN {X 0,Y 86.478,Z 505.707,A -85,B 0,C 180,E1 -27582.995,E2 -27582.995} C_VEL
LIN {X 0,Y 86.467,Z 505.708,A -85,B 0,C 180,E1 -27589.441,E2 -27589.441} C_VEL
LIN {X 0,Y 86.544,Z 505.704,A -85,B 0,C 180,E1 -27595.358,E2 -27595.358} C_VEL
LIN {X 0,Y 86.587,Z 505.699,A -85,B 0,C 180,E1 -27603.234,E2 -27603.234} C_VEL
LIN {X 0,Y 86.647,Z 505.688,A -85,B 0,C 180,E1 -27611.378,E2 -27611.378} C_VEL
LIN {X 0,Y 86.933,Z 505.648,A -85,B 0,C 180,E1 -27615.964,E2 -27615.964} C_VEL
LIN {X 0,Y 87.086,Z 505.637,A -85,B 0,C 180,E1 -27620.712,E2 -27620.712} C_VEL
LIN {X 0,Y 87.72,Z 505.559,A -85,B 0,C 180,E1 -27630.001,E2 -27630.001} C_VEL
LIN {X 0,Y 87.536,Z 505.573,A -85,B 0,C 180,E1 -27631.181,E2 -27631.181} C_VEL
LIN {X 0,Y 86.439,Z 505.712,A -85,B 0,C 180,E1 -27635.006,E2 -27635.006} C_VEL
LIN {X 0,Y 84.608,Z 505.946,A -85,B 0,C 180,E1 -27638.8,E2 -27638.8} C_VEL
LIN {X 0,Y 79.803,Z 506.541,A -85,B 0,C 180,E1 -27649.562,E2 -27649.562} C_VEL
LIN {X 0,Y 79.439,Z 506.575,A -85,B 0,C 180,E1 -27652.463,E2 -27652.463} C_VEL
LIN {X 0,Y 79.486,Z 506.582,A -85,B 0,C 180,E1 -27657.846,E2 -27657.846} C_VEL
LIN {X 0,Y 79.387,Z 506.589,A -85,B 0,C 180,E1 -27662.085,E2 -27662.085} C_VEL
LIN {X 0,Y 79.373,Z 506.591,A -85,B 0,C 180,E1 -27668.303,E2 -27668.303} C_VEL
LIN {X 0,Y 79.327,Z 506.603,A -85,B 0,C 180,E1 -27675.136,E2 -27675.136} C_VEL
LIN {X 0,Y 79.069,Z 506.636,A -85,B 0,C 180,E1 -27683.128,E2 -27683.128} C_VEL
LIN {X 0,Y 78.803,Z 506.66,A -85,B 0,C 180,E1 -27687.648,E2 -27687.648} C_VEL
LIN {X 0,Y 79.725,Z 506.699,A -85,B 0,C 180,E1 -27701.391,E2 -27701.391} C_VEL
LIN {X 0,Y 82.768,Z 520.819,A -85,B 0,C 180,E1 -27705.555,E2 -27705.555} C_VEL
LIN {X 0,Y 82.127,Z 529.965,A -85,B 0,C 180,E1 -27709.522,E2 -27709.522} C_VEL
LIN {X 0,Y 81.482,Z 541.537,A -85,B 0,C 180,E1 -27715.671,E2 -27715.671} C_VEL
LIN {X 0,Y 81.492,Z 552.045,A -85,B 0,C 180,E1 -27722.471,E2 -27722.471} C_VEL
LIN {X 0,Y 81.886,Z 558.517,A -85,B 0,C 180,E1 -27727.396,E2 -27727.396} C_VEL
LIN {X 0,Y 83.409,Z 567.933,A -85,B 0,C 180,E1 -27735.892,E2 -27735.892} C_VEL
LIN {X 0,Y 86.27,Z 575.726,A -85,B 0,C 180,E1 -27744.036,E2 -27744.036} C_VEL
LIN {X 0,Y 92.899,Z 584.484,A -85,B 0,C 180,E1 -27753.676,E2 -27753.676} C_VEL
LIN {X 0,Y 101.458,Z 591.211,A -85,B 0,C 180,E1 -27761.152,E2 -27761.152} C_VEL
LIN {X 0,Y 103.712,Z 592.635,A -85,B 0,C 180,E1 -27762.659,E2 -27762.659} C_VEL
LIN {X 0,Y 103.992,Z 592.982,A -85,B 0,C 180,E1 -27764.026,E2 -27764.026} C_VEL
LIN {X 0,Y 93.826,Z 588.023,A -85,B 0,C 180,E1 -27773.184,E2 -27773.184} C_VEL
LIN {X 0,Y 87.694,Z 582.107,A -85,B 0,C 180,E1 -27783.452,E2 -27783.452} C_VEL
LIN {X 0,Y 85.413,Z 574.154,A -85,B 0,C 180,E1 -27795.708,E2 -27795.708} C_VEL
LIN {X 0,Y 85.737,Z 569.299,A -85,B 0,C 180,E1 -27801.752,E2 -27801.752} C_VEL
LIN {X 0,Y 85.38,Z 565.382,A -85,B 0,C 180,E1 -27805.278,E2 -27805.278} C_VEL
LIN {X 0,Y 84.376,Z 556.378,A -85,B 0,C 180,E1 -27811.773,E2 -27811.773} C_VEL
LIN {X 0,Y 84.144,Z 547.324,A -85,B 0,C 180,E1 -27817.197,E2 -27817.197} C_VEL
LIN {X 0,Y 81.771,Z 536.343,A -85,B 0,C 180,E1 -27821.778,E2 -27821.778} C_VEL
LIN {X 0,Y 79.76,Z 523.042,A -85,B 0,C 180,E1 -27826.508,E2 -27826.508} C_VEL
LIN {X 0,Y 78.833,Z 509.5,A -85,B 0,C 180,E1 -27830.549,E2 -27830.549} C_VEL
LIN {X 0,Y 78.777,Z 506.668,A -85,B 0,C 180,E1 -27831.421,E2 -27831.421} C_VEL
LIN {X 0,Y 79.216,Z 506.616,A -85,B 0,C 180,E1 -27842.162,E2 -27842.162} C_VEL
LIN {X 0,Y 80.061,Z 506.513,A -85,B 0,C 180,E1 -27847.914,E2 -27847.914} C_VEL
LIN {X 0,Y 79.908,Z 506.527,A -85,B 0,C 180,E1 -27855.284,E2 -27855.284} C_VEL
LIN {X 0,Y 79.547,Z 506.568,A -85,B 0,C 180,E1 -27862.669,E2 -27862.669} C_VEL
LIN {X 0,Y 79.485,Z 506.575,A -85,B 0,C 180,E1 -27872.151,E2 -27872.151} C_VEL
LIN {X 0,Y 79.515,Z 506.573,A -85,B 0,C 180,E1 -27879.297,E2 -27879.297} C_VEL
LIN {X 0,Y 79.841,Z 506.539,A -85,B 0,C 180,E1 -27885.527,E2 -27885.527} C_VEL
LIN {X 0,Y 80.001,Z 506.512,A -85,B 0,C 180,E1 -27889.882,E2 -27889.882} C_VEL
LIN {X 0,Y 80.654,Z 506.435,A -85,B 0,C 180,E1 -27900.001,E2 -27900.001} C_VEL
LIN {X 0,Y 80.001,Z 506.519,A -85,B 0,C 180,E1 -27910.12,E2 -27910.12} C_VEL
LIN {X 0,Y 79.766,Z 506.539,A -85,B 0,C 180,E1 -27915.328,E2 -27915.328} C_VEL
LIN {X 0,Y 79.523,Z 506.578,A -85,B 0,C 180,E1 -27920.703,E2 -27920.703} C_VEL
LIN {X 0,Y 79.483,Z 506.584,A -85,B 0,C 180,E1 -27927.845,E2 -27927.845} C_VEL
LIN {X 0,Y 79.378,Z 506.589,A -85,B 0,C 180,E1 -27932.09,E2 -27932.09} C_VEL
LIN {X 0,Y 79.366,Z 506.598,A -85,B 0,C 180,E1 -27938.307,E2 -27938.307} C_VEL
LIN {X 0,Y 79.411,Z 506.593,A -85,B 0,C 180,E1 -27945.075,E2 -27945.075} C_VEL
LIN {X 0,Y 79.395,Z 506.592,A -85,B 0,C 180,E1 -27952.816,E2 -27952.816} C_VEL
LIN {X 0,Y 79.386,Z 506.589,A -85,B 0,C 180,E1 -27957.916,E2 -27957.916} C_VEL
LIN {X 0,Y 79.527,Z 506.579,A -85,B 0,C 180,E1 -27963.778,E2 -27963.778} C_VEL
LIN {X 0,Y 79.515,Z 506.574,A -85,B 0,C 180,E1 -27969.296,E2 -27969.296} C_VEL
LIN {X 0,Y 79.827,Z 506.535,A -85,B 0,C 180,E1 -27975.573,E2 -27975.573} C_VEL
LIN {X 0,Y 79.969,Z 506.522,A -85,B 0,C 180,E1 -27979.877,E2 -27979.877} C_VEL
LIN {X 0,Y 80.647,Z 506.44,A -85,B 0,C 180,E1 -27990.001,E2 -27990.001} C_VEL
LIN {X 0,Y 79.971,Z 506.522,A -85,B 0,C 180,E1 -28000.124,E2 -28000.124} C_VEL
LIN {X 0,Y 79.746,Z 506.548,A -85,B 0,C 180,E1 -28005.331,E2 -28005.331} C_VEL
LIN {X 0,Y 79.439,Z 506.575,A -85,B 0,C 180,E1 -28012.463,E2 -28012.463} C_VEL
LIN {X 0,Y 79.065,Z 506.635,A -85,B 0,C 180,E1 -28015.291,E2 -28015.291} C_VEL
LIN {X 0,Y 77.654,Z 506.811,A -85,B 0,C 180,E1 -28019.498,E2 -28019.498} C_VEL
LIN {X 0,Y 74.403,Z 507.216,A -85,B 0,C 180,E1 -28026.677,E2 -28026.677} C_VEL
LIN {X 0,Y 72.419,Z 507.464,A -85,B 0,C 180,E1 -28032.874,E2 -28032.874} C_VEL
LIN {X 0,Y 72.107,Z 507.494,A -85,B 0,C 180,E1 -28036.103,E2 -28036.103} C_VEL
LIN {X 0,Y 72.062,Z 507.507,A -85,B 0,C 180,E1 -28041.282,E2 -28041.282} C_VEL
LIN {X 0,Y 71.611,Z 507.565,A -85,B 0,C 180,E1 -28050.611,E2 -28050.611} C_VEL
LIN {X 0,Y 72.935,Z 507.399,A -85,B 0,C 180,E1 -28062.835,E2 -28062.835} C_VEL
LIN {X 0,Y 73.078,Z 507.6,A -85,B 0,C 180,E1 -28063.118,E2 -28063.118} C_VEL
LIN {X 0,Y 76.067,Z 520.872,A -85,B 0,C 180,E1 -28067.323,E2 -28067.323} C_VEL
LIN {X 0,Y 75.18,Z 534.087,A -85,B 0,C 180,E1 -28073.962,E2 -28073.962} C_VEL
LIN {X 0,Y 74.979,Z 543.898,A -85,B 0,C 180,E1 -28079.999,E2 -28079.999} C_VEL
LIN {X 0,Y 75.648,Z 554.574,A -85,B 0,C 180,E1 -28088.01,E2 -28088.01} C_VEL
LIN {X 0,Y 77.262,Z 564.579,A -85,B 0,C 180,E1 -28097.195,E2 -28097.195} C_VEL
LIN {X 0,Y 81.637,Z 574.807,A -85,B 0,C 180,E1 -28108.26,E2 -28108.26} C_VEL
LIN {X 0,Y 87.453,Z 581.887,A -85,B 0,C 180,E1 -28116.088,E2 -28116.088} C_VEL
LIN {X 0,Y 95.369,Z 588.361,A -85,B 0,C 180,E1 -28123.053,E2 -28123.053} C_VEL
LIN {X 0,Y 94.381,Z 588.07,A -85,B 0,C 180,E1 -28125.193,E2 -28125.193} C_VEL
LIN {X 0,Y 85.622,Z 582.531,A -85,B 0,C 180,E1 -28134.93,E2 -28134.93} C_VEL
LIN {X 0,Y 80.539,Z 575.484,A -85,B 0,C 180,E1 -28146.878,E2 -28146.878} C_VEL
LIN {X 0,Y 79.649,Z 567.861,A -85,B 0,C 180,E1 -28158.041,E2 -28158.041} C_VEL
LIN {X 0,Y 79.755,Z 565.454,A -85,B 0,C 180,E1 -28160.968,E2 -28160.968} C_VEL
LIN {X 0,Y 79.048,Z 560.855,A -85,B 0,C 180,E1 -28164.899,E2 -28164.899} C_VEL
LIN {X 0,Y 77.986,Z 551.084,A -85,B 0,C 180,E1 -28171.918,E2 -28171.918} C_VEL
LIN {X 0,Y 77.674,Z 545.172,A -85,B 0,C 180,E1 -28175.571,E2 -28175.571} C_VEL
LIN {X 0,Y 74.74,Z 532.895,A -85,B 0,C 180,E1 -28180.839,E2 -28180.839} C_VEL
LIN {X 0,Y 72.739,Z 519.411,A -85,B 0,C 180,E1 -28185.885,E2 -28185.885} C_VEL
LIN {X 0,Y 71.937,Z 507.515,A -85,B 0,C 180,E1 -28189.715,E2 -28189.715} C_VEL
LIN {X 0,Y 72.55,Z 507.443,A -85,B 0,C 180,E1 -28205.536,E2 -28205.536} C_VEL
LIN {X 0,Y 72.881,Z 507.408,A -85,B 0,C 180,E1 -28209.517,E2 -28209.517} C_VEL
LIN {X 0,Y 72.651,Z 507.435,A -85,B 0,C 180,E1 -28217.38,E2 -28217.38} C_VEL
LIN {X 0,Y 72.4,Z 507.461,A -85,B 0,C 180,E1 -28224.379,E2 -28224.379} C_VEL
LIN {X 0,Y 72.392,Z 507.458,A -85,B 0,C 180,E1 -28230.961,E2 -28230.961} C_VEL
LIN {X 0,Y 72.395,Z 507.466,A -85,B 0,C 180,E1 -28237.151,E2 -28237.151} C_VEL
LIN {X 0,Y 72.736,Z 507.425,A -85,B 0,C 180,E1 -28245.066,E2 -28245.066} C_VEL
LIN {X 0,Y 72.885,Z 507.397,A -85,B 0,C 180,E1 -28248.882,E2 -28248.882} C_VEL
LIN {X 0,Y 73.581,Z 507.316,A -85,B 0,C 180,E1 -28260.001,E2 -28260.001} C_VEL
LIN {X 0,Y 72.886,Z 507.406,A -85,B 0,C 180,E1 -28271.12,E2 -28271.12} C_VEL
LIN {X 0,Y 72.587,Z 507.437,A -85,B 0,C 180,E1 -28276.887,E2 -28276.887} C_VEL
LIN {X 0,Y 72.4,Z 507.46,A -85,B 0,C 180,E1 -28282.849,E2 -28282.849} C_VEL
LIN {X 0,Y 72.377,Z 507.469,A -85,B 0,C 180,E1 -28289.083,E2 -28289.083} C_VEL
LIN {X 0,Y 72.295,Z 507.478,A -85,B 0,C 180,E1 -28295.683,E2 -28295.683} C_VEL
LIN {X 0,Y 72.261,Z 507.477,A -85,B 0,C 180,E1 -28302.909,E2 -28302.909} C_VEL
LIN {X 0,Y 72.302,Z 507.47,A -85,B 0,C 180,E1 -28311.046,E2 -28311.046} C_VEL
LIN {X 0,Y 72.302,Z 507.479,A -85,B 0,C 180,E1 -28314.323,E2 -28314.323} C_VEL
LIN {X 0,Y 72.376,Z 507.464,A -85,B 0,C 180,E1 -28320.954,E2 -28320.954} C_VEL
LIN {X 0,Y 72.396,Z 507.459,A -85,B 0,C 180,E1 -28327.151,E2 -28327.151} C_VEL
LIN {X 0,Y 72.723,Z 507.421,A -85,B 0,C 180,E1 -28335.111,E2 -28335.111} C_VEL
LIN {X 0,Y 72.86,Z 507.405,A -85,B 0,C 180,E1 -28338.878,E2 -28338.878} C_VEL
LIN {X 0,Y 73.573,Z 507.321,A -85,B 0,C 180,E1 -28350.001,E2 -28350.001} C_VEL
LIN {X 0,Y 72.861,Z 507.405,A -85,B 0,C 180,E1 -28361.124,E2 -28361.124} C_VEL
LIN {X 0,Y 72.576,Z 507.444,A -85,B 0,C 180,E1 -28366.889,E2 -28366.889} C_VEL
LIN {X 0,Y 72.396,Z 507.459,A -85,B 0,C 180,E1 -28372.85,E2 -28372.85} C_VEL
LIN {X 0,Y 72.379,Z 507.463,A -85,B 0,C 180,E1 -28379.082,E2 -28379.082} C_VEL
LIN {X 0,Y 72.302,Z 507.479,A -85,B 0,C 180,E1 -28385.678,E2 -28385.678} C_VEL
LIN {X 0,Y 72.216,Z 507.489,A -85,B 0,C 180,E1 -28392.942,E2 -28392.942} C_VEL
LIN {X 0,Y 72.107,Z 507.494,A -85,B 0,C 180,E1 -28396.103,E2 -28396.103} C_VEL
LIN {X 0,Y 71.707,Z 507.549,A -85,B 0,C 180,E1 -28399.202,E2 -28399.202} C_VEL
LIN {X 0,Y 70.071,Z 507.761,A -85,B 0,C 180,E1 -28403.798,E2 -28403.798} C_VEL
LIN {X 0,Y 65.223,Z 508.365,A -85,B 0,C 180,E1 -28416.916,E2 -28416.916} C_VEL
LIN {X 0,Y 65.511,Z 508.321,A -85,B 0,C 180,E1 -28422.217,E2 -28422.217} C_VEL
LIN {X 0,Y 66.483,Z 508.362,A -85,B 0,C 180,E1 -28425.184,E2 -28425.184} C_VEL
LIN {X 0,Y 69.254,Z 519.771,A -85,B 0,C 180,E1 -28429.03,E2 -28429.03} C_VEL
LIN {X 0,Y 68.718,Z 530.814,A -85,B 0,C 180,E1 -28434.865,E2 -28434.865} C_VEL
LIN {X 0,Y 68.748,Z 541.913,A -85,B 0,C 180,E1 -28442.196,E2 -28442.196} C_VEL
LIN {X 0,Y 69.63,Z 551.995,A -85,B 0,C 180,E1 -28450.173,E2 -28450.173} C_VEL
LIN {X 0,Y 71.29,Z 560.86,A -85,B 0,C 180,E1 -28458.686,E2 -28458.686} C_VEL
LIN {X 0,Y 75.349,Z 570.572,A -85,B 0,C 180,E1 -28469.319,E2 -28469.319} C_VEL
LIN {X 0,Y 83.82,Z 580.582,A -85,B 0,C 180,E1 -28480.364,E2 -28480.364} C_VEL
LIN {X 0,Y 87.972,Z 584.021,A -85,B 0,C 180,E1 -28484.027,E2 -28484.027} C_VEL
LIN {X 0,Y 79.219,Z 577.86,A -85,B 0,C 180,E1 -28494.532,E2 -28494.532} C_VEL
LIN {X 0,Y 74.448,Z 570.039,A -85,B 0,C 180,E1 -28507.814,E2 -28507.814} C_VEL
LIN {X 0,Y 73.958,Z 563.964,A -85,B 0,C 180,E1 -28516.821,E2 -28516.821} C_VEL
LIN {X 0,Y 73.97,Z 562.2,A -85,B 0,C 180,E1 -28519.045,E2 -28519.045} C_VEL
LIN {X 0,Y 72.744,Z 556.02,A -85,B 0,C 180,E1 -28524.455,E2 -28524.455} C_VEL
LIN {X 0,Y 71.65,Z 545.401,A -85,B 0,C 180,E1 -28532.107,E2 -28532.107} C_VEL
LIN {X 0,Y 71.178,Z 543.021,A -85,B 0,C 180,E1 -28533.431,E2 -28533.431} C_VEL
LIN {X 0,Y 67.744,Z 529.039,A -85,B 0,C 180,E1 -28539.705,E2 -28539.705} C_VEL
LIN {X 0,Y 65.657,Z 513.852,A -85,B 0,C 180,E1 -28545.559,E2 -28545.559} C_VEL
LIN {X 0,Y 65.269,Z 508.351,A -85,B 0,C 180,E1 -28547.409,E2 -28547.409} C_VEL
LIN {X 0,Y 65.005,Z 508.384,A -85,B 0,C 180,E1 -28562.722,E2 -28562.722} C_VEL
LIN {X 0,Y 65.818,Z 508.288,A -85,B 0,C 180,E1 -28569.842,E2 -28569.842} C_VEL
LIN {X 0,Y 65.476,Z 508.327,A -85,B 0,C 180,E1 -28579.908,E2 -28579.908} C_VEL
LIN {X 0,Y 65.284,Z 508.348,A -85,B 0,C 180,E1 -28589.453,E2 -28589.453} C_VEL
LIN {X 0,Y 65.247,Z 508.356,A -85,B 0,C 180,E1 -28594.479,E2 -28594.479} C_VEL
LIN {X 0,Y 65.636,Z 508.31,A -85,B 0,C 180,E1 -28604.507,E2 -28604.507} C_VEL
LIN {X 0,Y 65.776,Z 508.284,A -85,B 0,C 180,E1 -28607.662,E2 -28607.662} C_VEL
LIN {X 0,Y 66.505,Z 508.197,A -85,B 0,C 180,E1 -28620.001,E2 -28620.001} C_VEL
LIN {X 0,Y 65.784,Z 508.289,A -85,B 0,C 180,E1 -28632.339,E2 -28632.339} C_VEL
LIN {X 0,Y 65.391,Z 508.339,A -85,B 0,C 180,E1 -28638.811,E2 -28638.811} C_VEL
LIN {X 0,Y 65.241,Z 508.351,A -85,B 0,C 180,E1 -28645.526,E2 -28645.526} C_VEL
LIN {X 0,Y 65.196,Z 508.354,A -85,B 0,C 180,E1 -28652.617,E2 -28652.617} C_VEL
LIN {X 0,Y 65.19,Z 508.356,A -85,B 0,C 180,E1 -28661.006,E2 -28661.006} C_VEL
LIN {X 0,Y 65.213,Z 508.353,A -85,B 0,C 180,E1 -28669.713,E2 -28669.713} C_VEL
LIN {X 0,Y 65.256,Z 508.347,A -85,B 0,C 180,E1 -28679.498,E2 -28679.498} C_VEL
LIN {X 0,Y 65.241,Z 508.358,A -85,B 0,C 180,E1 -28684.476,E2 -28684.476} C_VEL
LIN {X 0,Y 65.627,Z 508.307,A -85,B 0,C 180,E1 -28694.544,E2 -28694.544} C_VEL
LIN {X 0,Y 65.757,Z 508.285,A -85,B 0,C 180,E1 -28697.658,E2 -28697.658} C_VEL
LIN {X 0,Y 66.495,Z 508.203,A -85,B 0,C 180,E1 -28710.001,E2 -28710.001} C_VEL
LIN {X 0,Y 65.758,Z 508.285,A -85,B 0,C 180,E1 -28722.343,E2 -28722.343} C_VEL
LIN {X 0,Y 65.383,Z 508.34,A -85,B 0,C 180,E1 -28728.813,E2 -28728.813} C_VEL
LIN {X 0,Y 65.242,Z 508.358,A -85,B 0,C 180,E1 -28735.525,E2 -28735.525} C_VEL
LIN {X 0,Y 65.2,Z 508.358,A -85,B 0,C 180,E1 -28742.614,E2 -28742.614} C_VEL
LIN {X 0,Y 65.166,Z 508.361,A -85,B 0,C 180,E1 -28750.978,E2 -28750.978} C_VEL
LIN {X 0,Y 64.992,Z 508.382,A -85,B 0,C 180,E1 -28759.546,E2 -28759.546} C_VEL
LIN {X 0,Y 64.573,Z 508.441,A -85,B 0,C 180,E1 -28770.543,E2 -28770.543} C_VEL
LIN {X 0,Y 65.511,Z 508.321,A -85,B 0,C 180,E1 -28782.217,E2 -28782.217} C_VEL
LIN {X 0,Y 65.343,Z 508.86,A -85,B 0,C 180,E1 -28784.358,E2 -28784.358} C_VEL
LIN {X 0,Y 63.904,Z 510.698,A -85,B 0,C 180,E1 -28786.796,E2 -28786.796} C_VEL
LIN {X 0,Y 61.726,Z 514.142,A -85,B 0,C 180,E1 -28789.368,E2 -28789.368} C_VEL
LIN {X 0,Y 60.483,Z 518.427,A -85,B 0,C 180,E1 -28792.012,E2 -28792.012} C_VEL
LIN {X 0,Y 60.715,Z 523.447,A -85,B 0,C 180,E1 -28794.571,E2 -28794.571} C_VEL
LIN {X 0,Y 62.293,Z 531.313,A -85,B 0,C 180,E1 -28798.773,E2 -28798.773} C_VEL
LIN {X 0,Y 62.433,Z 533.187,A -85,B 0,C 180,E1 -28799.982,E2 -28799.982} C_VEL
LIN {X 0,Y 63.025,Z 543.769,A -85,B 0,C 180,E1 -28808.011,E2 -28808.011} C_VEL
LIN {X 0,Y 64.1,Z 550.841,A -85,B 0,C 180,E1 -28814.281,E2 -28814.281} C_VEL
LIN {X 0,Y 66.395,Z 559.622,A -85,B 0,C 180,E1 -28823.386,E2 -28823.386} C_VEL
LIN {X 0,Y 70.697,Z 568.202,A -85,B 0,C 180,E1 -28833.144,E2 -28833.144} C_VEL
LIN {X 0,Y 78.014,Z 576.709,A -85,B 0,C 180,E1 -28842.504,E2 -28842.504} C_VEL
LIN {X 0,Y 79.792,Z 578.338,A -85,B 0,C 180,E1 -28844.799,E2 -28844.799} C_VEL
LIN {X 0,Y 71.611,Z 571.035,A -85,B 0,C 180,E1 -28857.331,E2 -28857.331} C_VEL
LIN {X 0,Y 68.54,Z 563.459,A -85,B 0,C 180,E1 -28870.15,E2 -28870.15} C_VEL
LIN {X 0,Y 68.323,Z 558.69,A -85,B 0,C 180,E1 -28876.923,E2 -28876.923} C_VEL
LIN {X 0,Y 66.917,Z 552.535,A -85,B 0,C 180,E1 -28882.456,E2 -28882.456} C_VEL
LIN {X 0,Y 65.631,Z 543.747,A -85,B 0,C 180,E1 -28889.232,E2 -28889.232} C_VEL
LIN {X 0,Y 64.321,Z 539.198,A -85,B 0,C 180,E1 -28891.672,E2 -28891.672} C_VEL
LIN {X 0,Y 60.998,Z 525.952,A -85,B 0,C 180,E1 -28897.863,E2 -28897.863} C_VEL
LIN {X 0,Y 59.058,Z 512.752,A -85,B 0,C 180,E1 -28903.33,E2 -28903.33} C_VEL
LIN {X 0,Y 58.708,Z 509.169,A -85,B 0,C 180,E1 -28904.753,E2 -28904.753} C_VEL
LIN {X 0,Y 57.812,Z 509.283,A -85,B 0,C 180,E1 -28921.685,E2 -28921.685} C_VEL
LIN {X 0,Y 58.292,Z 509.221,A -85,B 0,C 180,E1 -28927.072,E2 -28927.072} C_VEL
LIN {X 0,Y 58.557,Z 509.182,A -85,B 0,C 180,E1 -28933.937,E2 -28933.937} C_VEL
LIN {X 0,Y 58.204,Z 509.225,A -85,B 0,C 180,E1 -28942.863,E2 -28942.863} C_VEL
LIN {X 0,Y 58.17,Z 509.229,A -85,B 0,C 180,E1 -28951.102,E2 -28951.102} C_VEL
LIN {X 0,Y 58.526,Z 509.194,A -85,B 0,C 180,E1 -28963.876,E2 -28963.876} C_VEL
LIN {X 0,Y 58.824,Z 509.158,A -85,B 0,C 180,E1 -28973.139,E2 -28973.139} C_VEL
LIN {X 0,Y 59.398,Z 509.082,A -85,B 0,C 180,E1 -28980.001,E2 -28980.001} C_VEL
LIN {X 0,Y 58.825,Z 509.148,A -85,B 0,C 180,E1 -28986.863,E2 -28986.863} C_VEL
LIN {X 0,Y 58.538,Z 509.184,A -85,B 0,C 180,E1 -28996.167,E2 -28996.167} C_VEL
LIN {X 0,Y 58.152,Z 509.241,A -85,B 0,C 180,E1 -29008.911,E2 -29008.911} C_VEL
LIN {X 0,Y 58.158,Z 509.231,A -85,B 0,C 180,E1 -29012.232,E2 -29012.232} C_VEL
LIN {X 0,Y 58.035,Z 509.256,A -85,B 0,C 180,E1 -29017.266,E2 -29017.266} C_VEL
LIN {X 0,Y 58.021,Z 509.258,A -85,B 0,C 180,E1 -29026.618,E2 -29026.618} C_VEL
LIN {X 0,Y 58.039,Z 509.251,A -85,B 0,C 180,E1 -29032.739,E2 -29032.739} C_VEL
LIN {X 0,Y 58.161,Z 509.233,A -85,B 0,C 180,E1 -29037.768,E2 -29037.768} C_VEL
LIN {X 0,Y 58.153,Z 509.235,A -85,B 0,C 180,E1 -29041.092,E2 -29041.092} C_VEL
LIN {X 0,Y 58.519,Z 509.194,A -85,B 0,C 180,E1 -29053.908,E2 -29053.908} C_VEL
LIN {X 0,Y 58.801,Z 509.157,A -85,B 0,C 180,E1 -29063.136,E2 -29063.136} C_VEL
LIN {X 0,Y 59.386,Z 509.088,A -85,B 0,C 180,E1 -29070.001,E2 -29070.001} C_VEL
LIN {X 0,Y 58.803,Z 509.157,A -85,B 0,C 180,E1 -29076.865,E2 -29076.865} C_VEL
LIN {X 0,Y 58.519,Z 509.194,A -85,B 0,C 180,E1 -29086.094,E2 -29086.094} C_VEL
LIN {X 0,Y 58.153,Z 509.235,A -85,B 0,C 180,E1 -29098.909,E2 -29098.909} C_VEL
LIN {X 0,Y 58.161,Z 509.232,A -85,B 0,C 180,E1 -29102.234,E2 -29102.234} C_VEL
LIN {X 0,Y 58.025,Z 509.253,A -85,B 0,C 180,E1 -29107.273,E2 -29107.273} C_VEL
LIN {X 0,Y 57.954,Z 509.266,A -85,B 0,C 180,E1 -29113.312,E2 -29113.312} C_VEL
LIN {X 0,Y 57.888,Z 509.267,A -85,B 0,C 180,E1 -29116.757,E2 -29116.757} C_VEL
LIN {X 0,Y 57.688,Z 509.299,A -85,B 0,C 180,E1 -29122.471,E2 -29122.471} C_VEL
LIN {X 0,Y 57.519,Z 509.32,A -85,B 0,C 180,E1 -29130.741,E2 -29130.741} C_VEL
LIN {X 0,Y 59.447,Z 509.076,A -85,B 0,C 180,E1 -29146.322,E2 -29146.322} C_VEL
LIN {X 0,Y 60.018,Z 509.008,A -85,B 0,C 180,E1 -29147.745,E2 -29147.745} C_VEL
LIN {X 0,Y 62.374,Z 518.269,A -85,B 0,C 180,E1 -29151.086,E2 -29151.086} C_VEL
LIN {X 0,Y 62.685,Z 520.192,A -85,B 0,C 180,E1 -29151.943,E2 -29151.943} C_VEL
LIN {X 0,Y 62.424,Z 532.039,A -85,B 0,C 180,E1 -29159.193,E2 -29159.193} C_VEL
LIN {X 0,Y 62.433,Z 533.187,A -85,B 0,C 180,E1 -29159.982,E2 -29159.982} C_VEL
LIN {X 0,Y 61.99,Z 537.61,A -85,B 0,C 180,E1 -29163.564,E2 -29163.564} C_VEL
LIN {X 0,Y 60.97,Z 541.47,A -85,B 0,C 180,E1 -29167.68,E2 -29167.68} C_VEL
LIN {X 0,Y 59.352,Z 548.365,A -85,B 0,C 180,E1 -29176.985,E2 -29176.985} C_VEL
LIN {X 0,Y 59.68,Z 551.939,A -85,B 0,C 180,E1 -29181.646,E2 -29181.646} C_VEL
LIN {X 0,Y 60.05,Z 553.211,A -85,B 0,C 180,E1 -29183.091,E2 -29183.091} C_VEL
LIN {X 0,Y 63.305,Z 560.799,A -85,B 0,C 180,E1 -29191.825,E2 -29191.825} C_VEL
LIN {X 0,Y 71.303,Z 571.295,A -85,B 0,C 180,E1 -29203.626,E2 -29203.626} C_VEL
LIN {X 0,Y 71.976,Z 571.94,A -85,B 0,C 180,E1 -29204.325,E2 -29204.325} C_VEL
LIN {X 0,Y 71.448,Z 571.63,A -85,B 0,C 180,E1 -29206.483,E2 -29206.483} C_VEL
LIN {X 0,Y 64.857,Z 563.956,A -85,B 0,C 180,E1 -29220.097,E2 -29220.097} C_VEL
LIN {X 0,Y 62.994,Z 556.749,A -85,B 0,C 180,E1 -29232.132,E2 -29232.132} C_VEL
LIN {X 0,Y 62.911,Z 555.626,A -85,B 0,C 180,E1 -29233.782,E2 -29233.782} C_VEL
LIN {X 0,Y 61.221,Z 548.865,A -85,B 0,C 180,E1 -29240.084,E2 -29240.084} C_VEL
LIN {X 0,Y 59.947,Z 541.8,A -85,B 0,C 180,E1 -29245.797,E2 -29245.797} C_VEL
LIN {X 0,Y 55.763,Z 528.417,A -85,B 0,C 180,E1 -29252.654,E2 -29252.654} C_VEL
LIN {X 0,Y 52.879,Z 513.441,A -85,B 0,C 180,E1 -29259.562,E2 -29259.562} C_VEL
LIN {X 0,Y 52.437,Z 509.948,A -85,B 0,C 180,E1 -29261.107,E2 -29261.107} C_VEL
LIN {X 0,Y 50.414,Z 510.199,A -85,B 0,C 180,E1 -29274.721,E2 -29274.721} C_VEL
LIN {X 0,Y 50.898,Z 510.138,A -85,B 0,C 180,E1 -29284.059,E2 -29284.059} C_VEL
LIN {X 0,Y 51.423,Z 510.071,A -85,B 0,C 180,E1 -29293.105,E2 -29293.105} C_VEL
LIN {X 0,Y 51.374,Z 510.084,A -85,B 0,C 180,E1 -29296.844,E2 -29296.844} C_VEL
LIN {X 0,Y 51.139,Z 510.115,A -85,B 0,C 180,E1 -29306.654,E2 -29306.654} C_VEL
LIN {X 0,Y 51.034,Z 510.128,A -85,B 0,C 180,E1 -29315.599,E2 -29315.599} C_VEL
LIN {X 0,Y 51.467,Z 510.074,A -85,B 0,C 180,E1 -29324.152,E2 -29324.152} C_VEL
LIN {X 0,Y 51.698,Z 510.044,A -85,B 0,C 180,E1 -29332.188,E2 -29332.188} C_VEL
LIN {X 0,Y 52.282,Z 509.967,A -85,B 0,C 180,E1 -29340.001,E2 -29340.001} C_VEL
LIN {X 0,Y 51.701,Z 510.036,A -85,B 0,C 180,E1 -29347.814,E2 -29347.814} C_VEL
LIN {X 0,Y 51.404,Z 510.074,A -85,B 0,C 180,E1 -29356.856,E2 -29356.856} C_VEL
LIN {X 0,Y 51.027,Z 510.119,A -85,B 0,C 180,E1 -29364.407,E2 -29364.407} C_VEL
LIN {X 0,Y 51.03,Z 510.12,A -85,B 0,C 180,E1 -29374.277,E2 -29374.277} C_VEL
LIN {X 0,Y 50.987,Z 510.134,A -85,B 0,C 180,E1 -29386.435,E2 -29386.435} C_VEL
LIN {X 0,Y 51.054,Z 510.122,A -85,B 0,C 180,E1 -29396.591,E2 -29396.591} C_VEL
LIN {X 0,Y 51.025,Z 510.125,A -85,B 0,C 180,E1 -29405.594,E2 -29405.594} C_VEL
LIN {X 0,Y 51.46,Z 510.072,A -85,B 0,C 180,E1 -29414.149,E2 -29414.149} C_VEL
LIN {X 0,Y 51.678,Z 510.047,A -85,B 0,C 180,E1 -29422.185,E2 -29422.185} C_VEL
LIN {X 0,Y 52.269,Z 509.975,A -85,B 0,C 180,E1 -29430.001,E2 -29430.001} C_VEL
LIN {X 0,Y 51.679,Z 510.047,A -85,B 0,C 180,E1 -29437.817,E2 -29437.817} C_VEL
LIN {X 0,Y 51.389,Z 510.084,A -85,B 0,C 180,E1 -29446.792,E2 -29446.792} C_VEL
LIN {X 0,Y 51.025,Z 510.125,A -85,B 0,C 180,E1 -29454.407,E2 -29454.407} C_VEL
LIN {X 0,Y 51.029,Z 510.128,A -85,B 0,C 180,E1 -29464.272,E2 -29464.272} C_VEL
LIN {X 0,Y 50.906,Z 510.144,A -85,B 0,C 180,E1 -29473.655,E2 -29473.655} C_VEL
LIN {X 0,Y 50.84,Z 510.146,A -85,B 0,C 180,E1 -29476.274,E2 -29476.274} C_VEL
LIN {X 0,Y 50.49,Z 510.186,A -85,B 0,C 180,E1 -29486.637,E2 -29486.637} C_VEL
LIN {X 0,Y 52.713,Z 509.919,A -85,B 0,C 180,E1 -29508.462,E2 -29508.462} C_VEL
LIN {X 0,Y 53.844,Z 509.819,A -85,B 0,C 180,E1 -29511.2,E2 -29511.2} C_VEL
LIN {X 0,Y 56.225,Z 518.665,A -85,B 0,C 180,E1 -29514.621,E2 -29514.621} C_VEL
LIN {X 0,Y 56.329,Z 529.575,A -85,B 0,C 180,E1 -29521.786,E2 -29521.786} C_VEL
LIN {X 0,Y 57.01,Z 538.744,A -85,B 0,C 180,E1 -29529.042,E2 -29529.042} C_VEL
LIN {X 0,Y 58.608,Z 547.84,A -85,B 0,C 180,E1 -29537.444,E2 -29537.444} C_VEL
LIN {X 0,Y 60.05,Z 553.211,A -85,B 0,C 180,E1 -29543.091,E2 -29543.091} C_VEL
LIN {X 0,Y 60.447,Z 555.403,A -85,B 0,C 180,E1 -29546.195,E2 -29546.195} C_VEL
LIN {X 0,Y 60.274,Z 557.852,A -85,B 0,C 180,E1 -29552.147,E2 -29552.147} C_VEL
LIN {X 0,Y 60.709,Z 560.137,A -85,B 0,C 180,E1 -29558.205,E2 -29558.205} C_VEL
LIN {X 0,Y 61.983,Z 562.083,A -85,B 0,C 180,E1 -29561.26,E2 -29561.26} C_VEL
LIN {X 0,Y 64.762,Z 565.294,A -85,B 0,C 180,E1 -29564.859,E2 -29564.859} C_VEL
LIN {X 0,Y 63.729,Z 564.371,A -85,B 0,C 180,E1 -29568.571,E2 -29568.571} C_VEL
LIN {X 0,Y 59.006,Z 557.282,A -85,B 0,C 180,E1 -29581.547,E2 -29581.547} C_VEL
LIN {X 0,Y 57.831,Z 552.005,A -85,B 0,C 180,E1 -29590.475,E2 -29590.475} C_VEL
LIN {X 0,Y 55.66,Z 545.01,A -85,B 0,C 180,E1 -29597.233,E2 -29597.233} C_VEL
LIN {X 0,Y 54.401,Z 539.708,A -85,B 0,C 180,E1 -29601.642,E2 -29601.642} C_VEL
LIN {X 0,Y 49.863,Z 526.569,A -85,B 0,C 180,E1 -29608.523,E2 -29608.523} C_VEL
LIN {X 0,Y 46.821,Z 512.769,A -85,B 0,C 180,E1 -29615.382,E2 -29615.382} C_VEL
LIN {X 0,Y 46.446,Z 510.696,A -85,B 0,C 180,E1 -29616.515,E2 -29616.515} C_VEL
LIN {X 0,Y 43.732,Z 511.03,A -85,B 0,C 180,E1 -29628.747,E2 -29628.747} C_VEL
LIN {X 0,Y 43.884,Z 511.011,A -85,B 0,C 180,E1 -29646.802,E2 -29646.802} C_VEL
LIN {X 0,Y 44.015,Z 511.003,A -85,B 0,C 180,E1 -29649.693,E2 -29649.693} C_VEL
LIN {X 0,Y 44.101,Z 510.986,A -85,B 0,C 180,E1 -29660.4,E2 -29660.4} C_VEL
LIN {X 0,Y 43.89,Z 511.007,A -85,B 0,C 180,E1 -29671.291,E2 -29671.291} C_VEL
LIN {X 0,Y 44.232,Z 510.969,A -85,B 0,C 180,E1 -29682.423,E2 -29682.423} C_VEL
LIN {X 0,Y 44.547,Z 510.929,A -85,B 0,C 180,E1 -29690.924,E2 -29690.924} C_VEL
LIN {X 0,Y 45.157,Z 510.854,A -85,B 0,C 180,E1 -29700.002,E2 -29700.002} C_VEL
LIN {X 0,Y 44.553,Z 510.93,A -85,B 0,C 180,E1 -29709.078,E2 -29709.078} C_VEL
LIN {X 0,Y 44.194,Z 510.978,A -85,B 0,C 180,E1 -29718.547,E2 -29718.547} C_VEL
LIN {X 0,Y 43.844,Z 511.024,A -85,B 0,C 180,E1 -29728.745,E2 -29728.745} C_VEL
LIN {X 0,Y 43.805,Z 511.021,A -85,B 0,C 180,E1 -29739.925,E2 -29739.925} C_VEL
LIN {X 0,Y 43.846,Z 511.019,A -85,B 0,C 180,E1 -29753.272,E2 -29753.272} C_VEL
LIN {X 0,Y 43.845,Z 511.016,A -85,B 0,C 180,E1 -29761.259,E2 -29761.259} C_VEL
LIN {X 0,Y 44.23,Z 510.976,A -85,B 0,C 180,E1 -29772.442,E2 -29772.442} C_VEL
LIN {X 0,Y 44.531,Z 510.938,A -85,B 0,C 180,E1 -29780.92,E2 -29780.92} C_VEL
LIN {X 0,Y 45.143,Z 510.862,A -85,B 0,C 180,E1 -29790.001,E2 -29790.001} C_VEL
LIN {X 0,Y 44.532,Z 510.938,A -85,B 0,C 180,E1 -29799.081,E2 -29799.081} C_VEL
LIN {X 0,Y 44.155,Z 510.983,A -85,B 0,C 180,E1 -29808.563,E2 -29808.563} C_VEL
LIN {X 0,Y 43.844,Z 511.016,A -85,B 0,C 180,E1 -29818.745,E2 -29818.745} C_VEL
LIN {X 0,Y 43.826,Z 511.022,A -85,B 0,C 180,E1 -29826.694,E2 -29826.694} C_VEL
LIN {X 0,Y 43.762,Z 511.024,A -85,B 0,C 180,E1 -29829.972,E2 -29829.972} C_VEL
LIN {X 0,Y 43.49,Z 511.059,A -85,B 0,C 180,E1 -29839.727,E2 -29839.727} C_VEL
LIN {X 0,Y 43.348,Z 511.085,A -85,B 0,C 180,E1 -29850.894,E2 -29850.894} C_VEL
LIN {X 0,Y 46.103,Z 510.738,A -85,B 0,C 180,E1 -29871.23,E2 -29871.23} C_VEL
LIN {X 0,Y 47.887,Z 510.57,A -85,B 0,C 180,E1 -29875.487,E2 -29875.487} C_VEL
LIN {X 0,Y 50.067,Z 518.071,A -85,B 0,C 180,E1 -29878.552,E2 -29878.552} C_VEL
LIN {X 0,Y 50.659,Z 529.238,A -85,B 0,C 180,E1 -29886.971,E2 -29886.971} C_VEL
LIN {X 0,Y 52.056,Z 539.037,A -85,B 0,C 180,E1 -29895.664,E2 -29895.664} C_VEL
LIN {X 0,Y 53.867,Z 546.346,A -85,B 0,C 180,E1 -29903.041,E2 -29903.041} C_VEL
LIN {X 0,Y 56.883,Z 553.919,A -85,B 0,C 180,E1 -29911.674,E2 -29911.674} C_VEL
LIN {X 0,Y 61.983,Z 562.083,A -85,B 0,C 180,E1 -29921.26,E2 -29921.26} C_VEL
LIN {X 0,Y 62.293,Z 562.647,A -85,B 0,C 180,E1 -29922.794,E2 -29922.794} C_VEL
LIN {X 0,Y 61.862,Z 562.383,A -85,B 0,C 180,E1 -29925.026,E2 -29925.026} C_VEL
LIN {X 0,Y 60.433,Z 560.945,A -85,B 0,C 180,E1 -29928.031,E2 -29928.031} C_VEL
LIN {X 0,Y 54.759,Z 553.566,A -85,B 0,C 180,E1 -29937.176,E2 -29937.176} C_VEL
LIN {X 0,Y 54.339,Z 552.727,A -85,B 0,C 180,E1 -29938.645,E2 -29938.645} C_VEL
LIN {X 0,Y 53.03,Z 548.221,A -85,B 0,C 180,E1 -29946.572,E2 -29946.572} C_VEL
LIN {X 0,Y 50.361,Z 540.749,A -85,B 0,C 180,E1 -29953.792,E2 -29953.792} C_VEL
LIN {X 0,Y 49.775,Z 538.66,A -85,B 0,C 180,E1 -29955.694,E2 -29955.694} C_VEL
LIN {X 0,Y 45.139,Z 526.927,A -85,B 0,C 180,E1 -29962.039,E2 -29962.039} C_VEL
LIN {X 0,Y 41.128,Z 511.889,A -85,B 0,C 180,E1 -29969.999,E2 -29969.999} C_VEL
LIN {X 0,Y 40.994,Z 511.37,A -85,B 0,C 180,E1 -29970.306,E2 -29970.306} C_VEL
LIN {X 0,Y 37.752,Z 511.775,A -85,B 0,C 180,E1 -29980.728,E2 -29980.728} C_VEL
LIN {X 0,Y 36.633,Z 511.911,A -85,B 0,C 180,E1 -30005.137,E2 -30005.137} C_VEL
LIN {X 0,Y 36.92,Z 511.884,A -85,B 0,C 180,E1 -30010.413,E2 -30010.413} C_VEL
LIN {X 0,Y 36.972,Z 511.876,A -85,B 0,C 180,E1 -30019.495,E2 -30019.495} C_VEL
LIN {X 0,Y 36.863,Z 511.887,A -85,B 0,C 180,E1 -30025.115,E2 -30025.115} C_VEL
LIN {X 0,Y 37.062,Z 511.859,A -85,B 0,C 180,E1 -30041.463,E2 -30041.463} C_VEL
LIN {X 0,Y 37.339,Z 511.823,A -85,B 0,C 180,E1 -30049.153,E2 -30049.153} C_VEL
LIN {X 0,Y 38.016,Z 511.742,A -85,B 0,C 180,E1 -30060.002,E2 -30060.002} C_VEL
LIN {X 0,Y 37.35,Z 511.833,A -85,B 0,C 180,E1 -30070.848,E2 -30070.848} C_VEL
LIN {X 0,Y 37.08,Z 511.863,A -85,B 0,C 180,E1 -30078.62,E2 -30078.62} C_VEL
LIN {X 0,Y 36.723,Z 511.903,A -85,B 0,C 180,E1 -30095.042,E2 -30095.042} C_VEL
LIN {X 0,Y 36.726,Z 511.901,A -85,B 0,C 180,E1 -30100.055,E2 -30100.055} C_VEL
LIN {X 0,Y 36.727,Z 511.9,A -85,B 0,C 180,E1 -30109.948,E2 -30109.948} C_VEL
LIN {X 0,Y 36.726,Z 511.911,A -85,B 0,C 180,E1 -30114.965,E2 -30114.965} C_VEL
LIN {X 0,Y 37.057,Z 511.867,A -85,B 0,C 180,E1 -30131.498,E2 -30131.498} C_VEL
LIN {X 0,Y 37.328,Z 511.828,A -85,B 0,C 180,E1 -30139.149,E2 -30139.149} C_VEL
LIN {X 0,Y 38.001,Z 511.752,A -85,B 0,C 180,E1 -30150.001,E2 -30150.001} C_VEL
LIN {X 0,Y 37.329,Z 511.828,A -85,B 0,C 180,E1 -30160.853,E2 -30160.853} C_VEL
LIN {X 0,Y 37.057,Z 511.867,A -85,B 0,C 180,E1 -30168.504,E2 -30168.504} C_VEL
LIN {X 0,Y 36.713,Z 511.912,A -85,B 0,C 180,E1 -30185.052,E2 -30185.052} C_VEL
LIN {X 0,Y 36.679,Z 511.905,A -85,B 0,C 180,E1 -30189.962,E2 -30189.962} C_VEL
LIN {X 0,Y 36.421,Z 511.941,A -85,B 0,C 180,E1 -30200.525,E2 -30200.525} C_VEL
LIN {X 0,Y 36.479,Z 511.932,A -85,B 0,C 180,E1 -30217.334,E2 -30217.334} C_VEL
LIN {X 0,Y 38.13,Z 511.736,A -85,B 0,C 180,E1 -30229.377,E2 -30229.377} C_VEL
LIN {X 0,Y 42.397,Z 511.196,A -85,B 0,C 180,E1 -30241.17,E2 -30241.17} C_VEL
LIN {X 0,Y 44.238,Z 516.648,A -85,B 0,C 180,E1 -30243.414,E2 -30243.414} C_VEL
LIN {X 0,Y 45.272,Z 526.865,A -85,B 0,C 180,E1 -30251.726,E2 -30251.726} C_VEL
LIN {X 0,Y 47.129,Z 536.441,A -85,B 0,C 180,E1 -30260.741,E2 -30260.741} C_VEL
LIN {X 0,Y 49.229,Z 542.963,A -85,B 0,C 180,E1 -30267.709,E2 -30267.709} C_VEL
LIN {X 0,Y 52.239,Z 549.68,A -85,B 0,C 180,E1 -30275.455,E2 -30275.455} C_VEL
LIN {X 0,Y 58.444,Z 558.754,A -85,B 0,C 180,E1 -30286.178,E2 -30286.178} C_VEL
LIN {X 0,Y 57.4,Z 557.548,A -85,B 0,C 180,E1 -30289.551,E2 -30289.551} C_VEL
LIN {X 0,Y 54.339,Z 552.727,A -85,B 0,C 180,E1 -30298.645,E2 -30298.645} C_VEL
LIN {X 0,Y 53.153,Z 550.396,A -85,B 0,C 180,E1 -30301.722,E2 -30301.722} C_VEL
LIN {X 0,Y 50.892,Z 546.413,A -85,B 0,C 180,E1 -30304.639,E2 -30304.639} C_VEL
LIN {X 0,Y 45.11,Z 535.99,A -85,B 0,C 180,E1 -30309.541,E2 -30309.541} C_VEL
LIN {X 0,Y 39.477,Z 522.593,A -85,B 0,C 180,E1 -30316.486,E2 -30316.486} C_VEL
LIN {X 0,Y 36.243,Z 511.961,A -85,B 0,C 180,E1 -30322.294,E2 -30322.294} C_VEL
LIN {X 0,Y 32.859,Z 512.353,A -85,B 0,C 180,E1 -30329.999,E2 -30329.999} C_VEL
LIN {X 0,Y 29.251,Z 512.696,A -85,B 0,C 180,E1 -30358.719,E2 -30358.719} C_VEL
LIN {X 0,Y 29.774,Z 512.645,A -85,B 0,C 180,E1 -30375.082,E2 -30375.082} C_VEL
LIN {X 0,Y 29.603,Z 512.661,A -85,B 0,C 180,E1 -30391.655,E2 -30391.655} C_VEL
LIN {X 0,Y 29.883,Z 512.634,A -85,B 0,C 180,E1 -30400.174,E2 -30400.174} C_VEL
LIN {X 0,Y 30.114,Z 512.615,A -85,B 0,C 180,E1 -30406.506,E2 -30406.506} C_VEL
LIN {X 0,Y 30.833,Z 512.546,A -85,B 0,C 180,E1 -30420.002,E2 -30420.002} C_VEL
LIN {X 0,Y 30.127,Z 512.612,A -85,B 0,C 180,E1 -30433.493,E2 -30433.493} C_VEL
LIN {X 0,Y 29.89,Z 512.637,A -85,B 0,C 180,E1 -30439.864,E2 -30439.864} C_VEL
LIN {X 0,Y 29.509,Z 512.672,A -85,B 0,C 180,E1 -30448.449,E2 -30448.449} C_VEL
LIN {X 0,Y 29.542,Z 512.67,A -85,B 0,C 180,E1 -30465.54,E2 -30465.54} C_VEL
LIN {X 0,Y 29.497,Z 512.672,A -85,B 0,C 180,E1 -30481.543,E2 -30481.543} C_VEL
LIN {X 0,Y 29.865,Z 512.638,A -85,B 0,C 180,E1 -30490.279,E2 -30490.279} C_VEL
LIN {X 0,Y 30.106,Z 512.614,A -85,B 0,C 180,E1 -30496.502,E2 -30496.502} C_VEL
LIN {X 0,Y 30.818,Z 512.551,A -85,B 0,C 180,E1 -30510.001,E2 -30510.001} C_VEL
LIN {X 0,Y 30.107,Z 512.614,A -85,B 0,C 180,E1 -30523.501,E2 -30523.501} C_VEL
LIN {X 0,Y 29.865,Z 512.638,A -85,B 0,C 180,E1 -30529.721,E2 -30529.721} C_VEL
LIN {X 0,Y 29.491,Z 512.673,A -85,B 0,C 180,E1 -30538.467,E2 -30538.467} C_VEL
LIN {X 0,Y 29.323,Z 512.688,A -85,B 0,C 180,E1 -30555.976,E2 -30555.976} C_VEL
LIN {X 0,Y 29.13,Z 512.707,A -85,B 0,C 180,E1 -30571.146,E2 -30571.146} C_VEL
LIN {X 0,Y 35.245,Z 512.087,A -85,B 0,C 180,E1 -30604.402,E2 -30604.402} C_VEL
LIN {X 0,Y 37.477,Z 511.812,A -85,B 0,C 180,E1 -30608.466,E2 -30608.466} C_VEL
LIN {X 0,Y 39.085,Z 516.279,A -85,B 0,C 180,E1 -30610.357,E2 -30610.357} C_VEL
LIN {X 0,Y 40.908,Z 526.874,A -85,B 0,C 180,E1 -30620.095,E2 -30620.095} C_VEL
LIN {X 0,Y 44.308,Z 537.518,A -85,B 0,C 180,E1 -30631.106,E2 -30631.106} C_VEL
LIN {X 0,Y 48.762,Z 546.547,A -85,B 0,C 180,E1 -30641.534,E2 -30641.534} C_VEL
LIN {X 0,Y 52.489,Z 551.712,A -85,B 0,C 180,E1 -30647.972,E2 -30647.972} C_VEL
LIN {X 0,Y 48.694,Z 544.633,A -85,B 0,C 180,E1 -30661.553,E2 -30661.553} C_VEL
LIN {X 0,Y 45.597,Z 537.056,A -85,B 0,C 180,E1 -30668.936,E2 -30668.936} C_VEL
LIN {X 0,Y 45.11,Z 535.99,A -85,B 0,C 180,E1 -30669.541,E2 -30669.541} C_VEL
LIN {X 0,Y 43.271,Z 532.636,A -85,B 0,C 180,E1 -30670.6,E2 -30670.6} C_VEL
LIN {X 0,Y 39.542,Z 527.096,A -85,B 0,C 180,E1 -30669.836,E2 -30669.836} C_VEL
LIN {X 0,Y 35.905,Z 521.368,A -85,B 0,C 180,E1 -30668.568,E2 -30668.568} C_VEL
LIN {X 0,Y 34.225,Z 517.682,A -85,B 0,C 180,E1 -30669.359,E2 -30669.359} C_VEL
LIN {X 0,Y 32.334,Z 512.403,A -85,B 0,C 180,E1 -30672.201,E2 -30672.201} C_VEL
LIN {X 0,Y 28.709,Z 512.746,A -85,B 0,C 180,E1 -30678.288,E2 -30678.288} C_VEL
LIN {X 0,Y 22.351,Z 513.08,A -85,B 0,C 180,E1 -30709.393,E2 -30709.393} C_VEL
LIN {X 0,Y 22.195,Z 513.084,A -85,B 0,C 180,E1 -30729.292,E2 -30729.292} C_VEL
LIN {X 0,Y 22.354,Z 513.079,A -85,B 0,C 180,E1 -30741.043,E2 -30741.043} C_VEL
LIN {X 0,Y 22.834,Z 513.064,A -85,B 0,C 180,E1 -30762.077,E2 -30762.077} C_VEL
LIN {X 0,Y 23.6,Z 513.041,A -85,B 0,C 180,E1 -30780.003,E2 -30780.003} C_VEL
LIN {X 0,Y 22.842,Z 513.064,A -85,B 0,C 180,E1 -30797.923,E2 -30797.923} C_VEL
LIN {X 0,Y 22.199,Z 513.084,A -85,B 0,C 180,E1 -30819.29,E2 -30819.29} C_VEL
LIN {X 0,Y 22.195,Z 513.084,A -85,B 0,C 180,E1 -30830.71,E2 -30830.71} C_VEL
LIN {X 0,Y 22.813,Z 513.065,A -85,B 0,C 180,E1 -30852.059,E2 -30852.059} C_VEL
LIN {X 0,Y 23.588,Z 513.042,A -85,B 0,C 180,E1 -30870.002,E2 -30870.002} C_VEL
LIN {X 0,Y 22.812,Z 513.065,A -85,B 0,C 180,E1 -30887.946,E2 -30887.946} C_VEL
LIN {X 0,Y 22.081,Z 513.088,A -85,B 0,C 180,E1 -30909.539,E2 -30909.539} C_VEL
LIN {X 0,Y 21.951,Z 513.092,A -85,B 0,C 180,E1 -30920.178,E2 -30920.178} C_VEL
LIN {X 0,Y 22.497,Z 513.075,A -85,B 0,C 180,E1 -30941.793,E2 -30941.793} C_VEL
LIN {X 0,Y 30.378,Z 512.589,A -85,B 0,C 180,E1 -30973.374,E2 -30973.374} C_VEL
LIN {X 0,Y 33.498,Z 512.321,A -85,B 0,C 180,E1 -30977.946,E2 -30977.946} C_VEL
LIN {X 0,Y 34.66,Z 515.476,A -85,B 0,C 180,E1 -30979.237,E2 -30979.237} C_VEL
LIN {X 0,Y 37.843,Z 527.061,A -85,B 0,C 180,E1 -30990.71,E2 -30990.71} C_VEL
LIN {X 0,Y 41.392,Z 535.491,A -85,B 0,C 180,E1 -30999.545,E2 -30999.545} C_VEL
LIN {X 0,Y 46.539,Z 543.756,A -85,B 0,C 180,E1 -31009.029,E2 -31009.029} C_VEL
LIN {X 0,Y 45.861,Z 542.55,A -85,B 0,C 180,E1 -31012.193,E2 -31012.193} C_VEL
LIN {X 0,Y 44.957,Z 540.748,A -85,B 0,C 180,E1 -31015.744,E2 -31015.744} C_VEL
LIN {X 0,Y 41.966,Z 534.749,A -85,B 0,C 180,E1 -31021.334,E2 -31021.334} C_VEL
LIN {X 0,Y 35.608,Z 521.317,A -85,B 0,C 180,E1 -31027.515,E2 -31027.515} C_VEL
LIN {X 0,Y 34.225,Z 517.682,A -85,B 0,C 180,E1 -31029.359,E2 -31029.359} C_VEL
LIN {X 0,Y 32.853,Z 515.681,A -85,B 0,C 180,E1 -31030.946,E2 -31030.946} C_VEL
LIN {X 0,Y 30.162,Z 514.026,A -85,B 0,C 180,E1 -31033.884,E2 -31033.884} C_VEL
LIN {X 0,Y 26.212,Z 513.169,A -85,B 0,C 180,E1 -31038.927,E2 -31038.927} C_VEL
LIN {X 0,Y 14.353,Z 513.178,A -85,B 0,C 180,E1 -31094.71,E2 -31094.71} C_VEL
LIN {X 0,Y 15.196,Z 513.178,A -85,B 0,C 180,E1 -31112.457,E2 -31112.457} C_VEL
LIN {X 0,Y 15.329,Z 513.178,A -85,B 0,C 180,E1 -31116.475,E2 -31116.475} C_VEL
LIN {X 0,Y 16.271,Z 513.178,A -85,B 0,C 180,E1 -31140.004,E2 -31140.004} C_VEL
LIN {X 0,Y 15.288,Z 513.178,A -85,B 0,C 180,E1 -31163.165,E2 -31163.165} C_VEL
LIN {X 0,Y 15.109,Z 513.178,A -85,B 0,C 180,E1 -31167.725,E2 -31167.725} C_VEL
LIN {X 0,Y 15.069,Z 513.178,A -85,B 0,C 180,E1 -31202.204,E2 -31202.204} C_VEL
LIN {X 0,Y 15.258,Z 513.178,A -85,B 0,C 180,E1 -31207.114,E2 -31207.114} C_VEL
LIN {X 0,Y 16.256,Z 513.178,A -85,B 0,C 180,E1 -31230.003,E2 -31230.003} C_VEL
LIN {X 0,Y 15.243,Z 513.178,A -85,B 0,C 180,E1 -31252.749,E2 -31252.749} C_VEL
LIN {X 0,Y 15.021,Z 513.178,A -85,B 0,C 180,E1 -31257.901,E2 -31257.901} C_VEL
LIN {X 0,Y 14.76,Z 513.178,A -85,B 0,C 180,E1 -31291.561,E2 -31291.561} C_VEL
LIN {X 0,Y 22.393,Z 513.078,A -85,B 0,C 180,E1 -31338.288,E2 -31338.288} C_VEL
LIN {X 0,Y 30.565,Z 512.57,A -85,B 0,C 180,E1 -31349.483,E2 -31349.483} C_VEL
LIN {X 0,Y 31.339,Z 514.442,A -85,B 0,C 180,E1 -31350.301,E2 -31350.301} C_VEL
LIN {X 0,Y 35.171,Z 524.901,A -85,B 0,C 180,E1 -31360.496,E2 -31360.496} C_VEL
LIN {X 0,Y 39.642,Z 533.129,A -85,B 0,C 180,E1 -31368.889,E2 -31368.889} C_VEL
LIN {X 0,Y 40.355,Z 534.144,A -85,B 0,C 180,E1 -31371.306,E2 -31371.306} C_VEL
LIN {X 0,Y 38.733,Z 531.292,A -85,B 0,C 180,E1 -31372.7,E2 -31372.7} C_VEL
LIN {X 0,Y 31.685,Z 516.774,A -85,B 0,C 180,E1 -31377.93,E2 -31377.93} C_VEL
LIN {X 0,Y 30.019,Z 512.625,A -85,B 0,C 180,E1 -31379.693,E2 -31379.693} C_VEL
LIN {X 0,Y 21.825,Z 513.096,A -85,B 0,C 180,E1 -31391.213,E2 -31391.213} C_VEL
LIN {X 0,Y 14.853,Z 513.178,A -85,B 0,C 180,E1 -31438.236,E2 -31438.236} C_VEL
LIN {X 0,Y 14.353,Z 513.178,A -85,B 0,C 180,E1 -31454.71,E2 -31454.71} C_VEL
LIN {X 0,Y 13.832,Z 513.178,A -85,B 0,C 180,E1 -31463.129,E2 -31463.129} C_VEL
LIN {X 0,Y 12.18,Z 513.178,A -85,B 0,C 180,E1 -31474.158,E2 -31474.158} C_VEL
LIN {X 0,Y 9.536,Z 513.178,A -85,B 0,C 180,E1 -31491.579,E2 -31491.579} C_VEL
LIN {X 0,Y 8.037,Z 513.178,A -85,B 0,C 180,E1 -31512.07,E2 -31512.07} C_VEL
LIN {X 0,Y 7.778,Z 513.178,A -85,B 0,C 180,E1 -31525.388,E2 -31525.388} C_VEL
LIN {X 0,Y 7.768,Z 513.178,A -85,B 0,C 180,E1 -31564.812,E2 -31564.812} C_VEL
LIN {X 0,Y 8.679,Z 513.178,A -85,B 0,C 180,E1 -31590.005,E2 -31590.005} C_VEL
LIN {X 0,Y 7.723,Z 513.178,A -85,B 0,C 180,E1 -31614.477,E2 -31614.477} C_VEL
LIN {X 0,Y 7.646,Z 513.178,A -85,B 0,C 180,E1 -31656.814,E2 -31656.814} C_VEL
LIN {X 0,Y 25.347,Z 512.987,A -85,B 0,C 180,E1 -31721.178,E2 -31721.178} C_VEL
LIN {X 0,Y 29.238,Z 512.699,A -85,B 0,C 180,E1 -31722.886,E2 -31722.886} C_VEL
LIN {X 0,Y 30.063,Z 514.688,A -85,B 0,C 180,E1 -31724.53,E2 -31724.53} C_VEL
LIN {X 0,Y 30.069,Z 514.72,A -85,B 0,C 180,E1 -31725.476,E2 -31725.476} C_VEL
LIN {X 0,Y 29.05,Z 512.713,A -85,B 0,C 180,E1 -31725.915,E2 -31725.915} C_VEL
LIN {X 0,Y 21.797,Z 513.097,A -85,B 0,C 180,E1 -31729.843,E2 -31729.843} C_VEL
LIN {X 0,Y 7.69,Z 513.178,A -85,B 0,C 180,E1 -31793.962,E2 -31793.962} C_VEL
LIN {X 0,Y 7.788,Z 513.178,A -85,B 0,C 180,E1 -31834.465,E2 -31834.465} C_VEL
LIN {X 0,Y 8.705,Z 513.178,A -85,B 0,C 180,E1 -31860.008,E2 -31860.008} C_VEL
LIN {X 0,Y 8.037,Z 513.178,A -85,B 0,C 180,E1 -31872.07,E2 -31872.07} C_VEL
LIN {X 0,Y 7.776,Z 515.178,A -85,B 0,C 180,E1 -31886.478,E2 -31886.478} C_VEL
LIN {X 0,Y 7.776,Z 600,A -85,B 0,C 180,E1 -31886.478,E2 -31886.478} C_VEL
LIN {X 0,Y 7.776,Z 600,A -85,B 0,C 180,E1 -31886.478,E2 -31886.478}

QRS_NEXT_CUT()

QRS_NEXT()
QRS_HOME()

END
